FUNCTION_BLOCK FB_Cylinder IMPLEMENTS I_Cylinder
VAR_INPUT
	bAtBasePos		AT %I*	: BOOL;		// Hardware input signal: cylinder is at base position
	bAtWorkPos		AT %I*	: BOOL;		// Hardware input signal: cylinder is at work position
END_VAR
VAR_OUTPUT
	bMoveToWork		AT %Q*	: BOOL;		// Hardware output signal to move cylinder to work position
END_VAR

// =========================================================
;
// =========================================================

PROPERTY PUBLIC bState_AtBasePos : BOOL
GET
bState_AtBasePos := bAtBasePos;
END_GET
END_PROPERTY

PROPERTY PUBLIC bState_AtWorkPos : BOOL
GET
bState_AtWorkPos := bAtWorkPos;
END_GET
END_PROPERTY

PROPERTY PUBLIC bState_MoveToWork : BOOL
GET
bState_MoveToWork := bMoveToWork;
END_GET
END_PROPERTY

METHOD MoveToBase
VAR_INPUT
END_VAR
// =========================================================
	
StateMachine(	bBasePosReq := TRUE,
				bWorkPosReq	:= FALSE );
							
// =========================================================
END_METHOD

METHOD MoveToWork
VAR_INPUT
END_VAR
// =========================================================
	
StateMachine(	bBasePosReq := FALSE,
				bWorkPosReq	:= TRUE );
								
// =========================================================
END_METHOD

METHOD Reset
VAR_INPUT
END_VAR
// =========================================================

bMoveToWork := FALSE;

// =========================================================
END_METHOD

METHOD PROTECTED StateMachine
VAR_INPUT
	bBasePosReq		: BOOL;
	bWorkPosReq		: BOOL;
END_VAR
// =========================================================
// Base or work position requested
		
	IF bWorkPosReq THEN
		bMoveToWork := TRUE;
	END_IF
	
	IF bBasePosReq OR NOT bWorkPosReq THEN
		bMoveToWork := FALSE;
	END_IF

// =========================================================
END_METHOD

END_FUNCTION_BLOCK

// ---- 01_Submodules/Cylinder/POUs/FB_CylinderDiag.TcPOU
(* FB_CylinderDiag	- number of control signals:
							one direction is controllable
					- type of feedback signal:
							feedback in base and work position
					- with position diagnosis						*)
					
FUNCTION_BLOCK FB_CylinderDiag EXTENDS FB_Cylinder
VAR_INPUT
	tTimeOut 	 		: TIME;					// Time for watchdog that monitores if cylinder reaches base/work position
	fVibrationSensor	AT %I*	: LREAL;		// Hardware input signal: cylinder vibration
	fPressureSensor		AT %I*	: LREAL;		// Hardware input signal: cylinder pressure
END_VAR
VAR_OUTPUT
	bError				: BOOL;			// Error signal (diagnosed from position watchdog)
	sErrorMsg			: STRING;		// Error message
END_VAR
VAR
	fbTriggerError		: R_TRIG;		// Trigger to recognize rising edge of error
	bErrorMove			: BOOL;			// Move error
	fbTimerWatchDog		: TON;			// Watchdog timer for monitoring if cylinder reaches base/work position
END_VAR

// =========================================================
;
// =========================================================

METHOD PROTECTED Diag
VAR_INPUT
END_VAR
// =========================================================
// Timer starts when cylinder is not in base and work position
	
	IF NOT bAtBasePos AND NOT bAtWorkPos THEN
		fbTimerWatchDog(IN := TRUE,
						PT := tTimeOut);
	ELSE
		fbTimerWatchDog(IN := FALSE,
						PT := tTimeOut);
	END_IF

// =========================================================
// Error if cylinder does not reach base or work position
	
	fbTriggerError(CLK := fbTimerWatchDog.Q);
	
	bError := fbTimerWatchDog.Q;
	
	IF fbTriggerError.Q THEN
		bErrorMove := bMoveToWork;
	END_IF
	
	IF bError THEN
		IF bErrorMove = bMoveToWork THEN
			IF bMoveToWork THEN
				sErrorMsg := 'Work position not reached';
			ELSE
				sErrorMsg := 'Base position not reached';
			END_IF
		ELSE
			bError := FALSE;
			sErrorMsg := '';
		END_IF
	ELSE
		sErrorMsg := '';
	END_IF

// =========================================================
END_METHOD

METHOD Reset
VAR_INPUT
END_VAR
// =========================================================

// Calling method Reset of base class FB_Cylinder via 'SUPER^.'
SUPER^.Reset();		

// Reset error
bError 		:= FALSE;
sErrorMsg 	:= '';

// =========================================================
END_METHOD

METHOD PROTECTED StateMachine
VAR_INPUT
	bBasePosReq		: BOOL;
	bWorkPosReq		: BOOL;
END_VAR
// =========================================================

IF NOT bError THEN
	// Calling method StateMachine of base class FB_Cylinder via 'SUPER^.'
	SUPER^.StateMachine(bBasePosReq := bBasePosReq,
						bWorkPosReq	:= bWorkPosReq );
	
	// Diagnosis
	Diag();
END_IF

// =========================================================
END_METHOD

END_FUNCTION_BLOCK

// ---- 01_Submodules/Cylinder/POUs/FB_CylinderTemp.TcPOU
(* FB_CylinderTemp	- number of control signals:
							one direction is controllable
					- type of feedback signal:
							feedback in base and work position
					- with temperature signal					*)

FUNCTION_BLOCK FB_CylinderTemp EXTENDS FB_Cylinder
VAR_INPUT
	fTempCurrent	AT %I*	: LREAL;		// Hardware input signal: cylinder temperature
END_VAR

// =========================================================
;
// =========================================================

END_FUNCTION_BLOCK

// ---- 01_Submodules/Cylinder/POUs/FB_CylinderTempDiag.TcPOU
(* FB_CylinderTempDiag		- number of control signals:
									one direction is controllable
							- type of feedback signal:
									feedback in base and work position
							- with temperature diagnosis					*)

FUNCTION_BLOCK FB_CylinderTempDiag EXTENDS FB_CylinderTemp
VAR_INPUT
	fTempMax		AT %I*	: LREAL;		// Global input signal: maximal allowed cylinder temperature for temperature monitoring
	fTempMin		AT %I*	: LREAL;		// Global input signal: minimal allowed cylinder temperature for temperature monitoring
END_VAR
VAR_OUTPUT
	bError					: BOOL;			// Error signal (diagnosed from temperature monitoring)
	sErrorMsg				: STRING;		// Error message
END_VAR

// =========================================================
;
// =========================================================

METHOD PROTECTED StateMachine
VAR_INPUT
	bBasePosReq		: BOOL;
	bWorkPosReq		: BOOL;
END_VAR
// =========================================================

IF NOT bError THEN
	// Calling method StateMachine of base class FB_Cylinder via 'SUPER^.'
	SUPER^.StateMachine(bBasePosReq := bBasePosReq,
						bWorkPosReq	:= bWorkPosReq );
	
	// Diagnosis
	Diag();
END_IF

// =========================================================
END_METHOD

METHOD Reset
VAR_INPUT
END_VAR
// =========================================================
	
// Calling method Reset of base class FB_Cylinder via 'SUPER^.'
SUPER^.Reset();			

// Reset error
bError 		:= FALSE;
sErrorMsg 	:= '';

// =========================================================
END_METHOD

METHOD PROTECTED Diag
VAR_INPUT
END_VAR
// =========================================================
// Error if temperatur of cylinder is not in accepted interval
	
	bError := NOT (fTempCurrent >= fTempMin AND fTempCurrent <= fTempMax);
	
	IF bError THEN
		IF fTempCurrent > fTempMax THEN
			sErrorMsg := 'Temperature above maximum';
		ELSE
			sErrorMsg := 'Temperature below minimum';
		END_IF
	ELSE
		sErrorMsg := '';
	END_IF

// =========================================================
END_METHOD

END_FUNCTION_BLOCK

// ---- 01_Submodules/Cylinder/POUs/FB_CylinderTempRecord.TcPOU
(* FB_CylinderTempRecord	- number of control signals:
									one direction is controllable
							- type of feedback signal:
									feedback in base and work position
							- with temperature recording for data analysis		*)

FUNCTION_BLOCK FB_CylinderTempRecord EXTENDS FB_CylinderTemp
VAR_INPUT
	bRecordStart		: BOOL;						// Signal to start the temperature recording
	tIntervalTime		: TIME;						// Time of intervals to record the temperature 
END_VAR
VAR_OUTPUT
	bRecordDone			: BOOL;						// True if the temperature recording is done
	aTemps				: ARRAY[1..100] OF LREAL;	// Array with recorded temperatures
END_VAR
VAR
	fbTimerInterval		: TON;						// Timer to control the recording interval
	nIndex				: INT;						// Index to handle temperature array
END_VAR

// =========================================================
;
// =========================================================

METHOD Record
VAR_INPUT
END_VAR
// =========================================================
// Recording array filled
	
	bRecordDone := (nIndex = 100);

// =========================================================
// Recording temperatures
	
	IF bRecordStart AND NOT bRecordDone AND NOT fbTimerInterval.Q THEN
		fbTimerInterval(IN := TRUE,
						PT := tIntervalTime );
	END_IF
	
	IF fbTimerInterval.Q THEN
		fbTimerInterval(IN := FALSE);
		
		nIndex 			:= nIndex + 1;
		aTemps[nIndex] 	:= fTempCurrent;
	END_IF

// =========================================================
END_METHOD

METHOD Reset
VAR_INPUT
END_VAR
// =========================================================

// Calling method Reset of base class FB_Cylinder via 'SUPER^.'
SUPER^.Reset();

// Reset temperature array
FOR nIndex := 1 TO 100 BY 1 DO
	aTemps[nIndex] := 0;
END_FOR

// Reset index
nIndex := 0;

// =========================================================
END_METHOD

END_FUNCTION_BLOCK

// ---- 02_Subsystems/FB_SortingModule.TcPOU
// Module to select via sensor, cylinder and axis
FUNCTION_BLOCK FB_SortingModule EXTENDS FB_Subsystem_Root
VAR_INPUT
	// =============== Cylinder buttons =============================================
	bButtonCylToWorkIn			: BOOL;							// Signal of button to move cylinder to work position
	bButtonCylToBaseIn			: BOOL;							// Signal of button to move cylinder to base position
END_VAR
VAR_OUTPUT
	// =============== Process information ==========================================
	bSelected					: BOOL;							// Gets true if one sorting process is done
	
	// =============== For movement simulation on visualization =====================
	bCylinderToWork				: BOOL;							// Simulation of cylinder movement to work position
	
	// =============== Error variables ==============================================
	bCylError					: BOOL;							// Error signal of cylinder
	sCylErrorMsg				: STRING;						// Error message of cylinder
	
	// =============== Temperature recording ========================================
	aTemps						: ARRAY[1..100] OF LREAL;		// Array with recorded temperatures of cylinder
	
	// =============== Button return signals ========================================
	bButtonCylToWorkOut			: BOOL;							// Processed signal for button to move cylinder to work position
	bButtonCylToBaseOut			: BOOL;							// Processed signal for button to move cylinder to base position
END_VAR
VAR
	// =============== Function block instance of sensor ============================	
	fbSensorDelay				: FB_SignalHandlingDelay;		// Sensor needed for sorting process
	
	// =============== Function block instances for cylinder ========================
	fbCylinder					: FB_Cylinder;					// Without diagnosis and temperature mode
	fbCylinderDiag				: FB_CylinderDiag;				// With diagnosis of states
	fbCylinderTemp				: FB_CylinderTemp;				// With temperature mode
	fbCylinderTempDiag			: FB_CylinderTempDiag;			// With diagnosis of temperature
	fbCylinderTempRecord		: FB_CylinderTempRecord;		// With record of temperatures
	
	// =============== Interface instance for cylinder ==============================
	ipCylinder					: I_Cylinder;					// Interface for flexible access to cylinder FBs
	
	// =============== Submodule parameters =========================================
	tTimeOutCylinder			: TIME;							// For cylinder with diagnosis: time in which the cylinder should reach base/work position
	tRecordIntervalCylinder		: TIME;							// Time of intervals to record the temperature of cylinder
	tSensorDelay				: TIME;							// Time to delay sensor signal (time between hardware and processed software signal)
	tMoveAxis					: TIME;							// Time to move axis
	
	// =============== Manual cylinder control ======================================
	fbButtonCylToWork			: FB_SignalHandlingIntern;		// To move cylinder manually to work position
	fbButtonCylToBase			: FB_SignalHandlingIntern;		// To move cylinder manually to base position

	// =============== Common variables =============================================
	fbTimerAxis					: TON;							// Timer to move axis in (semi) automatic mode	
	fbTriggerCylAtWork			: R_TRIG;						// Trigger to recognize rising edge of cylinder being at work position
	eStateAutoAxis				: E_StateSortingAutoAxis;		// State variable for automatic mode - process to move axis
	eStateAutoCylinder			: E_StateSortingAutoCylinder;	// State variable for automatic mode - process to move cylinder
END_VAR

// =========================================================
;
// =========================================================

METHOD Automatic
VAR_INPUT
END_VAR
// =========================================================
// Process of sorting boxes - axis movement

	fbTriggerCylAtWork(CLK := ipCylinder.bState_AtWorkPos);			// Accessing property of FB via interface instance

	CASE eStateAutoAxis OF
		
		// =========================================================
		E_StateSortingAutoAxis.WaitForCylinderAtWorkPos:
		
						IF fbTriggerCylAtWork.Q THEN
							fbTimerAxis(IN := TRUE,
										PT := tMoveAxis);
										
							eStateAutoAxis := E_StateSortingAutoAxis.MoveAxis;
						END_IF
		
		// =========================================================
		E_StateSortingAutoAxis.MoveAxis:
		
						fbTimerAxis();
						
						IF bHaltRequest THEN
							eStateAutoAxis := E_StateSortingAutoAxis.StopAxis;
						ELSIF fbTimerAxis.Q THEN
							fbTimerAxis(IN := FALSE);
							
							bSelected 		:= TRUE;
							eStateAutoAxis	:= E_StateSortingAutoAxis.StopAxis;
						ELSE
							fbAxis.MoveFw();
						END_IF
		
		
		// =========================================================
		E_StateSortingAutoAxis.StopAxis:
		
						bSelected := FALSE;
						
						IF NOT bHaltDone THEN
							Stop(bHalt := TRUE);
						ELSE
							Stop(bHalt := FALSE);
							
							eStateAutoAxis := E_StateSortingAutoAxis.WaitForCylinderAtWorkPos;
						END_IF
	END_CASE
	
// =========================================================
// Process of sorting boxes - cylinder movement

	CASE eStateAutoCylinder OF
		
		// =========================================================
		// Detecting a box
		E_StateSortingAutoCylinder.DetectBox:	
		
					ipCylinder.MoveToBase();								// Calling method of FB via interface instance
					
					IF fbSensorDelay.bOut THEN
						eStateAutoCylinder := E_StateSortingAutoCylinder.CylToWork;
					END_IF
			
		// =========================================================
		// Moving cylinder to work position
		E_StateSortingAutoCylinder.CylToWork:
		
					ipCylinder.MoveToWork();								// Calling method of FB via interface instance
					
					IF ipCylinder.bState_AtWorkPos THEN					// Accessing property of FB via interface instance
						eStateAutoCylinder := E_StateSortingAutoCylinder.CylToBase;
					END_IF
		
		// =========================================================
		// Moving cylinder back to base position
		E_StateSortingAutoCylinder.CylToBase:
		
					ipCylinder.MoveToBase();								// Calling method of FB via interface instance
					
					IF ipCylinder.bState_AtBasePos THEN					// Accessing property of FB via interface instance
						eStateAutoCylinder := E_StateSortingAutoCylinder.DetectBox;
					END_IF
	END_CASE

// =========================================================
END_METHOD

PROPERTY bState_CylinderAtBasePos : BOOL
GET
bState_CylinderAtBasePos := ipCylinder.bState_AtBasePos;
END_GET
END_PROPERTY

PROPERTY bState_CylinderAtWorkPos : BOOL
GET
bState_CylinderAtWorkPos := ipCylinder.bState_AtWorkPos;
END_GET
END_PROPERTY

METHOD CylinderOptions
VAR_INPUT
	bCylinderDiag		: BOOL;		// If true the cylinder has diagnosis functionality
	bCylinderTemp		: BOOL;		// IF true the cylinder has temperature functionality
	bCylinderRecord		: BOOL;		// If true the cylinder has recording functionality
END_VAR
// =========================================================
// Selecting cylinder

	// Checking variables to enable/disable diagnosis and temperature mode
	IF bCylinderDiag THEN
		IF bCylinderTemp THEN
			// ============== FB with diagnosis and temperature mode ==============
			bCylError 		:= fbCylinderTempDiag.bError;						// Assigning output variable of chosen FB to local output variable
			sCylErrorMsg 	:= fbCylinderTempDiag.sErrorMsg;
			ipCylinder		:= fbCylinderTempDiag;								// Assigning chosen FB instance to interface instance
		
		ELSE
			// ============== FB with diagnosis and without temperature mode ==============
			fbCylinderDiag.tTimeOut 	:= tTimeOutCylinder;					// Setting special data for selected FB
			bCylError 					:= fbCylinderDiag.bError;				// Assigning output variable of chosen FB to local output variable
			sCylErrorMsg 				:= fbCylinderDiag.sErrorMsg;		
			ipCylinder					:= fbCylinderDiag;						// Assigning chosen FB instance to interface instance
		END_IF
		
	ELSE
		bCylError 		:= FALSE;
		sCylErrorMsg 	:= '';
		
		IF bCylinderTemp THEN
			IF bCylinderRecord THEN
				// ============== FB without diagnosis and with temperature recording ==============
				fbCylinderTempRecord.tIntervalTime	:= tRecordIntervalCylinder;	// Time of record interval
				fbCylinderTempRecord.bRecordStart 	:= bComprAirEnabledLocal;	// Recording if compressed air is set
				
				fbCylinderTempRecord.Record();									// Calling method of function block FB_CylinderTempRecord
				
				aTemps		:= fbCylinderTempRecord.aTemps;						// Saving output variable
				ipCylinder 	:= fbCylinderTempRecord;							// Assigning chosen FB instance to interface instance
			ELSE
				// ============== FB without diagnosis and with temperature mode, but without recording ==============
				ipCylinder 	:= fbCylinderTemp; 									// Assigning chosen FB instance to interface instance
			END_IF
			
		ELSE
			// ============== FB without diagnosis and without temperature mode ==============
			ipCylinder := fbCylinder;											// Assigning chosen FB instance to interface instance					
		END_IF	
	END_IF
									
// =========================================================
END_METHOD

METHOD Enable
VAR_INPUT
	bComprAirEnabled		: BOOL;			// Enable of compressed air
	bAxisEnable				: BOOL;			// Enable of axis
	bSensorEnable			: BOOL;			// Enable of sensor
	bManualAxisEnable		: BOOL;			// Enable of manual axis control
END_VAR
// =========================================================
// Calling method Enable of base class FB_Module via 'SUPER^.'
		
	SUPER^.Enable(	bComprAirEnabled	:= bComprAirEnabled,
					bAxisEnable			:= bAxisEnable,
					bSensorEnable		:= bSensorEnable,
					bManualAxisEnable	:= bManualAxisEnable);

// =========================================================
// Sensor control
		
	fbSensorDelay.Enable(bEnable := bSensorEnable);

// =========================================================
// Cylinder control (accessing property of FB via interfaces intance)
		
	fbButtonCylToWork.Enable(bEnable := bManualCylinderEnable AND NOT ipCylinder.bState_AtWorkPos);
	fbButtonCylToBase.Enable(bEnable := bManualCylinderEnable AND NOT ipCylinder.bState_AtBasePos);
	
	fbButtonCylToBase.bInput := NOT fbButtonCylToWork.bInput;

// =========================================================
END_METHOD

METHOD InputOutput
VAR_INPUT
END_VAR
// =========================================================
// Calling method SetOutput of base class FB_Module via 'SUPER^.'
		
	SUPER^.InputOutput();

// =========================================================
// Sensor
		
	fbSensorDelay.SetOutput();

// =========================================================
// Cylinder buttons
		
	fbButtonCylToWork.SetOutput();
	fbButtonCylToBase.SetOutput();

// =========================================================
// Output variables for cylinder
		
	bCylinderToWork := ipCylinder.bState_MoveToWork;		// Accessing property of selected FB via interface instance

// =========================================================
// Buttons
		
	fbButtonCylToWork.bInput 	:= bButtonCylToWorkIn;
	fbButtonCylToBase.bInput	:= bButtonCylToBaseIn;
	bButtonCylToWorkOut 		:= fbButtonCylToWork.bOut;
	bButtonCylToBaseOut 		:= fbButtonCylToBase.bOut;

// =========================================================
END_METHOD

METHOD Maintenance
VAR_INPUT
END_VAR
// =========================================================
// Calling own method Manual of this class FB_SortingModule via 'THIS^.'
		
	THIS^.Manual();

// =========================================================
END_METHOD

METHOD Manual
VAR_INPUT
END_VAR
// =========================================================
// Calling method Manual of base class FB_Module via 'SUPER^.'
		
	SUPER^.Manual();

// =========================================================
// Manual cylinder control (Calling methods of FB via interface instance)
	
	// Cylinder to work position
	IF fbButtonCylToWork.bOut THEN
		ipCylinder.MoveToWork();
	// Cylinder to base position
	ELSIF fbButtonCylToBase.bOut THEN
		ipCylinder.MoveToBase();
	END_IF

// =========================================================
END_METHOD

METHOD Reset
VAR_INPUT
	bReset		: BOOL;				// True if machine is in state RESETTING
END_VAR
// =========================================================
// Calling action Reset of base class FB_Module via 'SUPER^.'
		
	SUPER^.Reset(bReset := bReset);

// =========================================================
// Resetting cylinder and axis
	
	IF fbTriggerResetStart.Q THEN
		bSelected := FALSE;
		
		fbTimerAxis(IN := FALSE);
		
		// Calling method of FB via interface instance
		ipCylinder.Reset();
	END_IF

// =========================================================
END_METHOD

METHOD PROTECTED ResetState
VAR_INPUT
END_VAR
// =========================================================

eStateAutoAxis		:= E_StateSortingAutoAxis.WaitForCylinderAtWorkPos;
eStateAutoCylinder 	:= E_StateSortingAutoCylinder.DetectBox;

// =========================================================
END_METHOD

METHOD Semiautomatic
VAR_INPUT
END_VAR
// =========================================================
// Calling own method Automatic of this class FB_SortingModule via 'THIS^.'
		
	THIS^.Automatic();				

// =========================================================
END_METHOD

METHOD Starting
VAR_INPUT
	bStarting		: BOOL;			// True if machine is in state STARTING
END_VAR
// =========================================================
// Setting time to delay sensor
		
	fbSensorDelay.tDelay := tSensorDelay;

// =========================================================
// Calling method Starting of base class FB_Module via 'SUPER^.'
		
	SUPER^.Starting(bStarting := bStarting);

// =========================================================
END_METHOD

PROPERTY tAxisMovement : TIME
GET
tAxisMovement := tMoveAxis;
END_GET
SET
tMoveAxis := tAxisMovement;
END_SET
END_PROPERTY

PROPERTY tDelayOfSensor : TIME
GET
tDelayOfSensor := tSensorDelay;
END_GET
SET
tSensorDelay := tDelayOfSensor;
END_SET
END_PROPERTY

PROPERTY tRecordIntervalOfCylinder : TIME
GET
tRecordIntervalOfCylinder := tRecordIntervalCylinder;
END_GET
SET
tRecordIntervalCylinder := tRecordIntervalOfCylinder;
END_SET
END_PROPERTY

PROPERTY tTimeOutOfCylinder : TIME
GET
tTimeOutOfCylinder := tTimeOutCylinder;
END_GET
SET
tTimeOutCylinder := tTimeOutOfCylinder;
END_SET
END_PROPERTY

END_FUNCTION_BLOCK

// ---- 01_Submodules/Signal handling/POUs/FB_SignalHandlingDelay.TcPOU
FUNCTION_BLOCK FB_SignalHandlingDelay EXTENDS FB_SignalHandling
VAR_INPUT
	tDelay				: TIME;			// Time to delay input signal (time between hardware and processed software signal)
END_VAR
VAR
	bStartProcessing	: BOOL;			// To start the processing/delay of input signal
	fbTimerDelay		: TON;			// Timer to control the processing/delay of input signal
END_VAR

// =========================================================
;
// =========================================================

METHOD SetOutput
VAR_INPUT
END_VAR
// =========================================================

IF bEnableLocal AND bInput THEN
	bStartProcessing := TRUE;
END_IF

IF bStartProcessing THEN
	fbTimerDelay(	IN := TRUE,
					PT := tDelay);
ELSE
	fbTimerDelay(	IN := FALSE);
END_IF

IF fbTimerDelay.Q THEN
	bStartProcessing := FALSE;
	
	fbTimerDelay(IN := FALSE);
	
	bOut := TRUE;
ELSE
	bOut := FALSE;
END_IF
			
// =========================================================
END_METHOD

END_FUNCTION_BLOCK

// ---- 05_Visu/FB_Visu.TcPOU
FUNCTION_BLOCK FB_Visu
VAR_INPUT
	// =============== Sensors to detect boxes ==================
	bBarrierSensor			AT %I*	: BOOL;						// True if barrier sensor detects a box
	bMetalSensor			AT %I*	: BOOL;						// True if metal sensor detects a metal box
	bPlasticSensor			AT %I*	: BOOL;						// True if plastic sensor detects a box
	
	// =============== Axis =====================================
	fAxisVelo						: LREAL;					// Axis velocity
	
	// =============== State of machine elements ================
	bComprAirEnabled				: BOOL;						// True if compressed air is enabled
	bPowerEnabled					: BOOL;						// True if power supply is enabled
	bMainAxisMoves					: BOOL;						// True if main axis is moving
	bMetalAxisMoves					: BOOL;						// True if metal axis is moving
	bPlasticAxisMoves				: BOOL;						// True if plastic axis is moving
	bClampToWork					: BOOL;						// True if clamp cylinder moves to work position
	bBarrierToWork					: BOOL;						// True if barrier cylinder moves to work position
	bMetalToWork					: BOOL;						// True if metal cylinder moves to work position
	bPlasticToWork					: BOOL;						// True if plastic cylinder moves to work position
	
	// =============== Error ====================================
	bError							: BOOL;						// True if modules have errors
	bClampError						: BOOL;						// True if clamp cylinder has an error
	sClampErrMsg					: STRING;					// Error message of clamp cylinder
	bMetalCylError					: BOOL;						// True if metal cylinder has an error
	sMetalErrMsg					: STRING;					// Error message of metal cylinder
	bPlasticCylError				: BOOL;						// True if plastic cylinder has an error
	sPlasticErrMsg					: STRING;					// Error message of plastic cylinder
	nMainAxisErrorId				: UDINT;					// Error id of main axis
	nMetalAxisErrorId				: UDINT;					// Error id of metal axis
	nPlasticAxisErrorId				: UDINT;					// Error id of plastic axis
	
	// =============== PS_PackML_StateMachine ===================
	bStarted						: BOOL;						// True if state machine is in state EXECUTE
	bStopped						: BOOL;						// True if state machine is in state STOPPED
	bReset							: BOOL;						// True if state machine is in state RESETTING
	bAborted						: BOOL;						// True if state machine is in state ABORTED
	bIdle							: BOOL;						// True if state machine is in state IDLE
	bAuto							: BOOL;						// True if state machine is in mode AUTOMATIC
	bSemi							: BOOL;						// True if state machine is in mode SEMIAUTOMATIC
	bManual							: BOOL;						// True if state machine is in mode MANUAL
	bMaintenance					: BOOL;						// True if state machine is in mode MAINTENANCE
	bStartButtonOff					: BOOL;						// To turn off start button

	// =============== Buttons of visualization - inputs ========
	// State buttons
	bButtonPowerIn					: BOOL;						// Input signal of power button
	bButtonComprAirIn				: BOOL;						// Input signal of compressed air button
	bButtonStartIn					: BOOL;						// Input signal of start button
	bButtonStopIn					: BOOL;						// Input signal of stop button
	bButtonResetIn					: BOOL;						// Input signal of reset button
	bButtonAbortIn					: BOOL;						// Input signal of abort button
	
	// Mode buttons
	bButtonAutoIn					: BOOL;						// Input signal of automatic button
	bButtonSemiIn					: BOOL;						// Input signal of semi-automatic button
	bButtonManuIn					: BOOL;						// Input signal of manual button
	bButtonMaintenanceIn			: BOOL;						// Input signal of maintenance button
	
	// Axis buttons
	bButtonMainFwIn					: BOOL;						// Input signal of button to move main axis forwards
	bButtonMainBwIn					: BOOL;						// Input signal of button to move main axis backwards
	bButtonMetalFwIn				: BOOL;						// Input signal of button to move metal axis forwards
	bButtonMetalBwIn				: BOOL;						// Input signal of button to move metal axis backwards
	bButtonPlasticFwIn				: BOOL;						// Input signal of button to move plastic axis forwards
	bButtonPlasticBwIn				: BOOL;						// Input signal of button to move plastic axis backwards
	
	// Cylinder buttons
	bButtonClampToWorkIn			: BOOL;						// Input signal of button to move clamp cylinder
	bButtonBarrierToWorkIn			: BOOL;						// Input signal of button to move barrier cylinder
	bButtonMetalToWorkIn			: BOOL;						// Input signal of button to move metal cylinder
	bButtonPlasticToWorkIn			: BOOL;						// Input signal of button to move plastic cylinder
END_VAR
VAR_OUTPUT
	fYClamp					AT %Q*	: LREAL;					// Y-Coordinate of clamp cylinder
	fYBarrier				AT %Q*	: LREAL;					// Y-Coordinate of barrier cylinder
	fYMetal					AT %Q*	: LREAL;					// Y-Coordinate of metal cylinder
	fYPlastic				AT %Q*	: LREAL;					// Y-Coordinate of plastic cylinder
	aBoxX					AT %Q*	: ARRAY[1..4] OF LREAL;		// X-Coordinates of boxes
	aBoxY					AT %Q*	: ARRAY[1..4] OF LREAL;		// Y-Coordinates of boxes
	
	// =============== Buttons of visualization - outputs =======
	// State buttons
	bButtonPowerOut					: BOOL;						// To turn on and off the machine
	bButtonComprAirOut				: BOOL;						// To enable compressed air
	bButtonStartOut					: BOOL;						// To change state into state START
	bButtonStopOut					: BOOL;						// To change state into state STOP
	bButtonResetOut					: BOOL;						// To change state into state RESET
	
	// Mode buttons
	bButtonAutoOut					: BOOL;						// To change mode into mode AUTOMATIC		
	bButtonSemiOut					: BOOL;						// To change mode into mode SEMI-AUTOMATIC	
	bButtonManuOut					: BOOL;						// To change mode into mode MANAUL	
	bButtonMaintenanceOut			: BOOL;						// To change mode into mode MAINTENANCE	
	
	// Axis buttons
	bButtonMainFwOut				: BOOL;						// To move main axis forwards
	bButtonMainBwOut				: BOOL;						// To move main axis backwards
	bButtonMetalFwOut				: BOOL;						// To move metal axis forwards
	bButtonMetalBwOut				: BOOL;						// To move metal axis backwards
	bButtonPlasticFwOut				: BOOL;						// To move plastic axis forwards
	bButtonPlasticBwOut				: BOOL;						// To move plastic axis backwards
	
	// Cylinder buttons
	bButtonClampToWorkOut			: BOOL;						// To move manually clamp cylinder to work position
	bButtonBarrierToWorkOut			: BOOL;						// To move manually barrier cylinder to work position
	bButtonMetalToWorkOut			: BOOL;						// To move manually metal cylinder to work position
	bButtonPlasticToWorkOut			: BOOL;						// To move manually plastic cylinder to work position
END_VAR
VAR
	// =============== Boxes movement ===========================
	nLastBox						: INT;						// Box on last position of main belt
	aBoxMetalMove					: ARRAY[1..4] OF BOOL;		// bBoxMetalMove[1] is true, if box 1 is moved by metal cylinder
	aBoxMetalFree					: ARRAY[1..4] OF BOOL;		// bBoxMetalFree[1] is true, if any box blockades the movement of box 1 on metal belt
	aBoxPlasticMove					: ARRAY[1..4] OF BOOL;		// bBoxPlasticMove[1] is true, if box 1 is moved by plastic cylinder
	aBoxPlasticFree					: ARRAY[1..4] OF BOOL;		// bBoxMetalFree[1] is true, if any box blockades the plastic belt
	aBoxMainBelt					: ARRAY[1..4] OF BOOL;		// bBoxMainBelt[1] is true, if box 1 is on main belt and has no obstacles, so box 1 is moved by main axis
	aBoxMetalBelt					: ARRAY[1..4] OF BOOL;		// aBoxMetalBelt[1] is true, if box 1 is on metal belt and has no obstacles, so box 1 is moved by metal axis
	aBoxPlasticBelt					: ARRAY[1..4] OF BOOL;		// aBoxPlasticBelt[1] is true, if box 1 is on plastic belt and has no obstacles, so box 1 is moved by plastic axis
	fMainVelo						: LREAL;					// Velocity of boxes on main belt
	fMetalVelo						: LREAL;					// Velocity of boxes on metal belt
	fPlasticVelo					: LREAL;					// Velocity of boxes on plastic belt
	bAccident						: BOOL;						// True if machine caused an accident
	nState							: INT;
	
	// =============== Message ==================================
	nMessages						: INT;						// Number of messages
	sMessageClamp					: STRING;					// Message of clamp cylinder
	sMessageMetalCyl				: STRING;					// Message of metal cylinder
	sMessagePlasticCyl				: STRING;					// Message of plastic cylinder
	sMessageMainAxis				: STRING;					// Message of main axis
	sMessageMetalAxis				: STRING;					// Message of metal axis
	sMessagePlasticAxis				: STRING;					// Message of plastic axis
	
	// =============== Axes movement ============================
	nAngleMain						: INT;						// Angle of main axis element
	nAngleMetal						: INT;						// Angle of metal axis element
	nAnglePlastic					: INT;						// Angle of plastic axis element
	fbTimerMainAxis					: TON;						// Timer for movement of main axis element
	fbTimerMetalAxis				: TON;						// Timer for movement of metal axis element
	fbTimerPlasticAxis				: TON;						// Timer for movement of plastic axis element
	tMoveAxis						: TIME := T#40MS;			// Time for movement of elements

	// =============== Color variables ==========================
	nButtonColorStart				: DWORD;					// Color of start button
	bButtonColorStart				: BOOL;						// To change color of start button
	nButtonColorStop				: DWORD;					// Color of stop button
	bButtonColorStop				: BOOL;						// To change color of stop button
	nButtonColorReset				: DWORD;					// Color of reset button
	bButtonColorReset				: BOOL;						// To change color of reset button
	nButtonColorAuto				: DWORD;					// Color of automatic button
	bButtonColorAuto				: BOOL;						// To change color of automatic button
	nButtonColorSemi				: DWORD;					// Color of semi-automatic button
	bButtonColorSemi				: BOOL;						// To change color of semi-automatic button
	nButtonColorManu				: DWORD;					// Color of manual button
	bButtonColorManu				: BOOL;						// To change color of manual button
	nButtonColorMaint				: DWORD;					// Color of maintenance button
	bButtonColorMaint				: BOOL;						// To change color of maintenance button
	nButtonColorClamp				: DWORD;					// Color of button to move clamp cylinder
	bButtonColorClamp				: BOOL;						// To change color of clamp button
	nButtonColorBarrier				: DWORD;					// Color of button to move barrier cylinder
	bButtonColorBarrier				: BOOL;						// To change color of barrier button
	nButtonColorMetalCyl			: DWORD;					// Color of button to move metal cylinder
	bButtonColorMetalCyl			: BOOL;						// To change color of metal cylinder button
	nButtonColorPlasticCyl			: DWORD;					// Color of button to move plastic cylinder
	bButtonColorPlasticCyl			: BOOL;						// To change color of plastic cylinder button
	nButtonColorMainFw				: DWORD;					// Color of button to move main axis forwards
	bButtonColorMainFw				: BOOL;						// To change color of button to move main axis fw.
	nButtonColorMainBw				: DWORD;					// Color of button to move main axis backwards
	bButtonColorMainBw				: BOOL;						// To change color of button to move main axis bw.
	nButtonColorMetalFw				: DWORD;					// Color of button to move metal axis forwards
	bButtonColorMetalFw				: BOOL;						// To change color of button to move metal axis fw.
	nButtonColorMetalBw				: DWORD;					// Color of button to move metal axis backwards
	bButtonColorMetalBw				: BOOL;						// To change color of button to move metal axis bw.
	nButtonColorPlasticFw			: DWORD;					// Color of button to move plastic axis forwards
	bButtonColorPlasticFw			: BOOL;						// To change color of button to move plastic axis fw.
	nButtonColorPlasticBw			: DWORD;					// Color of button to move plastic axis backwards
	bButtonColorPlasticBw			: BOOL;						// To change color of button to move plastic axis bw.
	nButtonColorComprAir			: DWORD;					// Color of button to enable/disable compressed air
	bButtonColorComprAir			: BOOL;						// To change color of button to control compressed air
	
	// ================= PPM calc ===========================================
	ctTotalCtr						: CTU;
	ctMetalCtr						: CTU;
	arrTotal						: ARRAY[0..9] OF DINT;
	arrMetal						: ARRAY[0..9] OF DINT;
	tmrPpm							: TON;
	
END_VAR
VAR CONSTANT
	// =============== Colors ===============================================
	cYellow 									: DWORD	:= 16#00FFFF80;		// Color code for yellow
	cGreen 										: DWORD	:= 16#0080FF00;		// Color code for green
	cPink 										: DWORD	:= 16#00FF8080;		// Color code for pink
	
	// =============== Velocities ===========================================
	cVelocityDenominator						: LREAL := 250.0;			// Velocity of visualization is a fraction of real axis velocity
	cAxisMovementSemiPlusAuto					: INT 	:= 2;				// Axis movement per cycle in mode Automatic and Semi Autoamtic
	cAxisMovementManual							: INT 	:= 1;				// Axis movement per cycle in mode Manual
	cClampMovement								: LREAL := 0.1;				// Cylinder movement per cycle for clamp cylinder
	cBarrierMovement							: LREAL := 1.0;				// Cylinder movement per cycle for barrier cylinder
	cMetalPlasticCylMovement					: LREAL := 1.0;				// Cylinder movement per cycle for metal and plastic cylinder
	
	// =============== Barrier, clamp, metal, plastic cylinder ==============
	cYClampCylStartPos							: LREAL := 0.0;				// Y-start-position of clamp cylinder (where movement starts)
	cYClampCylEndPos							: LREAL := 3.0;				// Y-end-position of clamp cylinder (where movement ends)
	cYBarrierCylStartPos						: LREAL := 0.0;				// Y-start-position of barrier cylinder (where movement starts)
	cYBarrierCylEndPos							: LREAL := 63.0;			// Y-end-position of barrier cylinder (where movement ends)
	cYMetalPlasticCylStartPos					: LREAL := 0.0;				// Y-start-position of metal and plastic cylinder (where movement starts)
	cYMetalPlasticCylEndPos						: LREAL := -73.0;			// Y-end-position of metal and plastic cylinder (where movement ends)
	
	// =============== Widths, distances ====================================
	cBoxWidth									: LREAL := 60.0;			// Width of a box in the visu
	cBarrierWidth								: LREAL := 30.0;			// Width of the barrier cylinder in the visu
	cDiffBarrierToStartOfMetalCyl				: LREAL := 191.0;			// Difference on visu from barrier to start of metal cylinder
	cDiffBarrierToEndOfMetalCyl					: LREAL := 261.0;			// Difference on visu from barrier to end of metal cylinder
	cDiffBarrierToStartOfPlasticCyl				: LREAL := 441.0;			// Difference on visu from barrier to start of plastic cylinder
	cYMetalPlasticCylOnMainBelt					: LREAL := -9.0;			// Y-Position of metal and plastic cylinder reaching the main belt
	cYBoxesOnMetalPlasticBelt_min				: LREAL := -65.0;			// Minimal Y-Position of boxes when being on metal or plastic belt
	cYBoxesOnMetalPlasticBelt_max				: LREAL := -140.0;			// Maximal Y-Position of boxes when being on metal or plastic belt
	
	// =============== Positions of boxes - main belt =======================
	cYforAllBoxesOnMainBelt						: LREAL := -5.0;			// Y-Position of boxes being on main belt
	cYforAllBoxesNotOnMainBelt					: LREAL := -60.0;			// Y-Position of boxes not being on main belt
	
	cYforAllBoxesStartPosMainBelt				: LREAL := 0.0;				// Y-Position of boxes when being on first position of main belt
	cXforAllBoxesStartPosMainBelt				: LREAL := -240.0;			// X-Position of boxes when being on first position of main belt
	cXforAllBoxesLastPossiblePosMainBelt		: LREAL := 461.0;			// Last possible X-position of boxes on main belt
	
	cXforAllBoxesCorrectPushMetalCyl_min		: LREAL := 180;				// Minimal X-Position of boxes when being pushed by metal cylinder to metal belt 
	cXforAllBoxesCorrectPushMetalCyl_max		: LREAL := 211;				// Maximal X-Position of boxes when being pushed by metal cylinder to metal belt 
	cXforAllBoxesIncorrectPushMetalCyl_min		: LREAL := 131;				// Minimal X-Position of boxes when being pushed by metal cylinder, but not pushed to metal belt
	cXforAllBoxesIncorrectPushMetalCyl_max		: LREAL := 261;				// Maximal X-Position of boxes when being pushed by metal cylinder, but not pushed to metal belt
	
	cXforAllBoxesCorrectPushPlasticCyl_min		: LREAL := 430;				// Minimal X-Position of boxes when being pushed by plastic cylinder to plastic belt 
	cXforAllBoxesCorrectPushPlasticCyl_max		: LREAL := 461;				// Minimal X-Position of boxes when being pushed by plastic cylinder to plastic belt 
	cXforAllBoxesIncorrectPushPlasticCyl_min	: LREAL := 381;				// Minimal X-Position of boxes when being pushed by plastic cylinder, but not pushed to plastic belt
	
	// Box 1
	cXforBox1_MainBelt_Diff2to1_min				: LREAL := 0.001;			// Minimal distance from box 2 to box 1 so that box 1 can be moved on main belt
	cXforBox1_MainBelt_Diff2to1_max				: LREAL := 119.99999;		// Maximal distance from box 2 to box 1 so that box 1 can be moved on main belt
	cXforBox1_MainBelt_Diff3to1_min				: LREAL := 60.001;			// Minimal distance from box 3 to box 1 so that box 1 can be moved on main belt
	cXforBox1_MainBelt_Diff3to1_max				: LREAL := 179.99999;		// Maximal distance from box 3 to box 1 so that box 1 can be moved on main belt
	cXforBox1_MainBelt_Diff4to1_min				: LREAL := 120.001;			// Minimal distance from box 4 to box 1 so that box 1 can be moved on main belt
	cXforBox1_MainBelt_Diff4to1_max				: LREAL := 239.99999;		// Maximal distance from box 4 to box 1 so that box 1 can be moved on main belt
	
	// Box 2
	cXforBox2_MainBelt_Diff1to2_min				: LREAL := -0.00001;		// Minimal distance from box 1 to box 2 so that box 2 can be moved on main belt
	cXforBox2_MainBelt_Diff1to2_max				: LREAL := -119.999;		// Maximal distance from box 1 to box 2 so that box 2 can be moved on main belt
	cXforBox2_MainBelt_Diff3to2_min				: LREAL := 119.99999;		// Minimal distance from box 3 to box 2 so that box 2 can be moved on main belt
	cXforBox2_MainBelt_Diff3to2_max				: LREAL := 0.001;			// Maximal distance from box 3 to box 2 so that box 2 can be moved on main belt
	cXforBox2_MainBelt_Diff4to2_min				: LREAL := 179.99999;		// Minimal distance from box 4 to box 2 so that box 2 can be moved on main belt
	cXforBox2_MainBelt_Diff4to2_max				: LREAL := 60.001;			// Maximal distance from box 4 to box 2 so that box 2 can be moved on main belt

	// Box 3
	cXforBox3_MainBelt_Diff1to3_min				: LREAL := -60.00001;		// Minimal distance from box 1 to box 3 so that box 3 can be moved on main belt
	cXforBox3_MainBelt_Diff1to3_max				: LREAL := -179.999;		// Maximal distance from box 1 to box 3 so that box 3 can be moved on main belt
	cXforBox3_MainBelt_Diff2to3_min				: LREAL := -0.00001;		// Minimal distance from box 2 to box 3 so that box 3 can be moved on main belt
	cXforBox3_MainBelt_Diff2to3_max				: LREAL := -119.999;		// Maximal distance from box 2 to box 3 so that box 3 can be moved on main belt
	cXforBox3_MainBelt_Diff4to3_min				: LREAL := 119.99999;		// Minimal distance from box 4 to box 3 so that box 3 can be moved on main belt
	cXforBox3_MainBelt_Diff4to3_max				: LREAL := 0.001;			// Maximal distance from box 4 to box 3 so that box 3 can be moved on main belt
	
	// Box 4
	cXforBox4_MainBelt_Diff1to4_min				: LREAL := -120.00001;		// Minimal distance from box 1 to box 4 so that box 4 can be moved on main belt
	cXforBox4_MainBelt_Diff1to4_max				: LREAL := -239.999;		// Maximal distance from box 1 to box 4 so that box 4 can be moved on main belt
	cXforBox4_MainBelt_Diff2to4_min				: LREAL := -60.00001;		// Minimal distance from box 2 to box 4 so that box 4 can be moved on main belt
	cXforBox4_MainBelt_Diff2to4_max				: LREAL := -179.999;		// Maximal distance from box 2 to box 4 so that box 4 can be moved on main belt
	cXforBox4_MainBelt_Diff3to4_min				: LREAL := -0.00001;		// Minimal distance from box 3 to box 4 so that box 4 can be moved on main belt
	cXforBox4_MainBelt_Diff3to4_max				: LREAL := -119.999;		// Maximal distance from box 3 to box 4 so that box 4 can be moved on main belt
	
	// =============== Positions of boxes - metal belt ======================
	// Box 1
	cXforBox1OnMetalBelt_min					: LREAL := 240;				// Minimal X-Position of box 1 when being on metal belt
	cXforBox1OnMetalBelt_max					: LREAL := 271;				// Maximal X-Position of box 1 when being on metal belt
	// Box 2
	cXforBox2OnMetalBelt_min					: LREAL := 300;				// Minimal X-Position of box 2 when being on metal belt
	cXforBox2OnMetalBelt_max					: LREAL := 331;				// Maximal X-Position of box 2 when being on metal belt
	// Box 3
	cXforBox3OnMetalBelt_min					: LREAL := 360;				// Minimal X-Position of box 3 when being on metal belt
	cXforBox3OnMetalBelt_max					: LREAL := 391;				// Maximal X-Position of box 3 when being on metal belt
	// Box 4
	cXforBox4OnMetalBelt_min					: LREAL := 420;				// Minimal X-Position of box 4 when being on metal belt
	cXforBox4OnMetalBelt_max					: LREAL := 451;				// Maximal X-Position of box 4 when being on metal belt
	
	// =============== Positions of boxes - plastic belt ====================
	// Box 1
	cXforBox1OnPlasticBelt_min					: LREAL := 470;				// Minimal X-Position of box 1 when being on plastic belt
	cXforBox1OnPlasticBelt_max					: LREAL := 521;				// Maximal X-Position of box 1 when being on plastic belt
	// Box 2
	cXforBox2OnPlasticBelt_min					: LREAL := 530;				// Minimal X-Position of box 2 when being on plastic belt
	cXforBox2OnPlasticBelt_max					: LREAL := 581;				// Maximal X-Position of box 2 when being on plastic belt
	// Box 3
	cXforBox3OnPlasticBelt_min					: LREAL := 590;				// Minimal X-Position of box 3 when being on plastic belt
	cXforBox3OnPlasticBelt_max					: LREAL := 641;				// Maximal X-Position of box 3 when being on plastic belt
	// Box 4
	cXforBox4OnPlasticBelt_min					: LREAL := 650;				// Minimal X-Position of box 4 when being on plastic belt
	cXforBox4OnPlasticBelt_max					: LREAL := 701;				// Maximal X-Position of box 4 when being on plastic belt
END_VAR

// =========================================================
// Resetting visu
	
	IF bReset THEN
		Reset();
	END_IF

// =========================================================
// Because of the visualisation size, the boxes velocity is a fraction of the axis velocity
	
	IF bAuto OR bSemi OR bButtonMainFwIn THEN
		fMainVelo := (fAxisVelo / cVelocityDenominator);
	ELSIF bButtonMainBwIn THEN
		fMainVelo := -(fAxisVelo / cVelocityDenominator);
	END_IF
	
	IF bAuto OR bSemi OR bButtonMetalFwIn THEN
		fMetalVelo := -(fAxisVelo / cVelocityDenominator);
	ELSIF bButtonMetalBwIn THEN
		fMetalVelo := (fAxisVelo / cVelocityDenominator);
	END_IF
	
	IF bAuto OR bSemi OR bButtonPlasticFwIn THEN
		fPlasticVelo := -(fAxisVelo / cVelocityDenominator);
	ELSIF bButtonPlasticBwIn THEN
		fPlasticVelo := (fAxisVelo / cVelocityDenominator);
	END_IF

// =========================================================
// In case of accident the power button is turned off
	
	IF bAccident THEN
		IF bButtonPowerOut THEN
			bButtonPowerOut := FALSE;
		END_IF
		
		IF bStopped THEN
			bAccident := FALSE;
		END_IF
	END_IF

// =========================================================
// Visuazation functions

	// Rotation of axis elements
	AxisRotation();
	
	// Buttons, order of boxes, error messages
	ButtonSignals();
	ButtonColors();
	LastBox();
	ErrorMessages();
	
	// Motion of cylinders
	Barrier_Clamp_Cyl();
	Metal_Plastic_Cyl();
	
	// Motion of boxes
	AxisMoveBoxes();
	CylinderMoveBoxes();

// =========================================================

// ==========================================================
// part per min calculation
tmrPpm(IN:=(NOT tmrPpm.Q), PT:=T#60S);
IF tmrPpm.Q THEN
	MEMCPY(ADR(arrTotal[1]), ADR(arrTotal[0]), SIZEOF(DINT) * 9);
	MEMCPY(ADR(arrMetal[1]), ADR(arrMetal[0]), SIZEOF(DINT) * 9);
END_IF
ctTotalCtr(CU:=bMetalToWork OR bPlasticToWork, CV=>arrTotal[0], RESET:=tmrPpm.Q);
ctMetalCtr(CU:=bMetalToWork, CV=>arrMetal[0], RESET:=tmrPpm.Q);

// ===========================================================

METHOD PRIVATE AxisMoveBoxes
VAR_INPUT
END_VAR
// =========================================================
// Checking traction standby on main belt
// bBoxMainBelt[1] is true, if box 1 is on main belt and has no obstacles, so box 1 is moved by main axis
		
	aBoxMainBelt[1] := 	// box 1 on main belt
						aBoxY[1] >= cYforAllBoxesOnMainBelt	
						// not previous to box 2											
						AND (	(aBoxX[2] - aBoxX[1] - fMainVelo) >= cXforBox1_MainBelt_Diff2to1_max
							OR 	(aBoxX[2] - aBoxX[1] - fMainVelo) <= cXforBox1_MainBelt_Diff2to1_min
							OR 	aBoxY[2] < cYforAllBoxesNotOnMainBelt)
						// not previous to box 3	
						AND (	(aBoxX[3] - aBoxX[1] - fMainVelo) >= cXforBox1_MainBelt_Diff3to1_max
							OR 	(aBoxX[3] - aBoxX[1]- fMainVelo) <= cXforBox1_MainBelt_Diff3to1_min
							OR 	aBoxY[3] < cYforAllBoxesNotOnMainBelt)
						// not previous to box 4
						AND (	(aBoxX[4] - aBoxX[1] - fMainVelo) >= cXforBox1_MainBelt_Diff4to1_max
							OR 	(aBoxX[4] - aBoxX[1]- fMainVelo) <= cXforBox1_MainBelt_Diff4to1_min
							OR	aBoxY[4] < cYforAllBoxesNotOnMainBelt);
						
	aBoxMainBelt[2] := 	// box 2 on main belt
						aBoxY[2] >= cYforAllBoxesOnMainBelt
						// not previous to box 1											
						AND (	(aBoxX[1] - aBoxX[2] - fMainVelo) >= cXforBox2_MainBelt_Diff1to2_min 
							OR 	(aBoxX[1] - aBoxX[2] - fMainVelo) <= cXforBox2_MainBelt_Diff1to2_max 
							OR 	aBoxY[1] < cYforAllBoxesNotOnMainBelt)
						// not previous to box 3											
						AND (	(aBoxX[3] - aBoxX[2] - fMainVelo) >= cXforBox2_MainBelt_Diff3to2_min 
							OR 	(aBoxX[3] - aBoxX[2] - fMainVelo) <= cXforBox2_MainBelt_Diff3to2_max 
							OR 	aBoxY[3] < cYforAllBoxesNotOnMainBelt)
						// not previous to box 4											
						AND (	(aBoxX[4] - aBoxX[2] - fMainVelo) >= cXforBox2_MainBelt_Diff4to2_min 
							OR 	(aBoxX[4] - aBoxX[2] - fMainVelo) <= cXforBox2_MainBelt_Diff4to2_max 
							OR 	aBoxY[4] < cYforAllBoxesNotOnMainBelt);
	
	aBoxMainBelt[3] := 	// box 3 on main belt
						aBoxY[3] >= cYforAllBoxesOnMainBelt
						// not previous to box 1											
						AND (	(aBoxX[1] - aBoxX[3] - fMainVelo) >= cXforBox3_MainBelt_Diff1to3_min
							OR 	(aBoxX[1] - aBoxX[3] - fMainVelo) <= cXforBox3_MainBelt_Diff1to3_max
							OR 	aBoxY[1] < cYforAllBoxesNotOnMainBelt)
						// not previous to box 2											
						AND (	(aBoxX[2] - aBoxX[3] - fMainVelo) >= cXforBox3_MainBelt_Diff2to3_min
							OR 	(aBoxX[2] - aBoxX[3] - fMainVelo) <= cXforBox3_MainBelt_Diff2to3_max 
							OR 	aBoxY[2] < cYforAllBoxesNotOnMainBelt)
						// not previous to box 4											
						AND (	(aBoxX[4] - aBoxX[3] - fMainVelo) >= cXforBox3_MainBelt_Diff4to3_min
							OR 	(aBoxX[4] - aBoxX[3] - fMainVelo) <= cXforBox3_MainBelt_Diff4to3_max
							OR 	aBoxY[4] < cYforAllBoxesNotOnMainBelt);
						
	aBoxMainBelt[4] := 	// box 4 on main belt
						aBoxY[4] >= cYforAllBoxesOnMainBelt
						// not previous to box 1											
						AND (	(aBoxX[1] - aBoxX[4] - fMainVelo) >= cXforBox4_MainBelt_Diff1to4_min
							OR 	(aBoxX[1] - aBoxX[4] - fMainVelo) <= cXforBox4_MainBelt_Diff1to4_max
							OR 	aBoxY[1] < cYforAllBoxesNotOnMainBelt)
						// not previous to box 2											
						AND (	(aBoxX[2] - aBoxX[4] - fMainVelo) >= cXforBox4_MainBelt_Diff2to4_min
							OR 	(aBoxX[2] - aBoxX[4] - fMainVelo) <= cXforBox4_MainBelt_Diff2to4_max
							OR 	aBoxY[2] < cYforAllBoxesNotOnMainBelt)
						// not previous to box 3											
						AND (	(aBoxX[3] - aBoxX[4] - fMainVelo) >= cXforBox4_MainBelt_Diff3to4_min
							OR 	(aBoxX[3] - aBoxX[4] - fMainVelo) <= cXforBox4_MainBelt_Diff3to4_max
							OR 	aBoxY[3] < cYforAllBoxesNotOnMainBelt);
					
// =========================================================
// Motion of boxes on main belt - forwards
					
	IF bMainAxisMoves AND (bAuto OR bSemi OR bButtonMainFwIn) THEN
		FOR nState := 1 TO 4 BY 1 DO
			IF aBoxMainBelt[nState] THEN	
				// not previous to moving metal cylinder
				IF aBoxX[nState] >= (cBoxWidth*nState + cBarrierWidth) AND aBoxX[nState] < (cBoxWidth*nState + cDiffBarrierToEndOfMetalCyl - 1) THEN
					// Metal cylinder over main belt
					IF fYMetal <= cYMetalPlasticCylOnMainBelt THEN
						IF aBoxX[nState] < (cBoxWidth*nState + cDiffBarrierToStartOfMetalCyl - cBoxWidth + 0.25)
						AND aBoxX[nState] > (cBoxWidth*nState + cDiffBarrierToStartOfMetalCyl - cBoxWidth - 0.15) THEN
							aBoxX[nState] := cBoxWidth*nState + cDiffBarrierToStartOfMetalCyl - cBoxWidth;
						ELSIF aBoxX[nState] <= (cBoxWidth*nState + cDiffBarrierToStartOfMetalCyl - cBoxWidth - 0.15) THEN
							aBoxX[nState] := aBoxX[nState] + fMainVelo;
						END_IF
					// Metal cylinder not over main belt
					ELSE
						aBoxX[nState] := aBoxX[nState] + fMainVelo;
					END_IF
				END_IF
				
				// not previous to moving plastic cylinder
				IF aBoxX[nState] >= (cBoxWidth*nState + cDiffBarrierToEndOfMetalCyl - 1) THEN
					// Plastic cylinder over main belt
					IF fYPlastic <= cYMetalPlasticCylOnMainBelt THEN
						IF aBoxX[nState] < (cBoxWidth*nState + cDiffBarrierToStartOfPlasticCyl - cBoxWidth + 0.25)
						AND aBoxX[nState] > (cBoxWidth*nState + cDiffBarrierToStartOfPlasticCyl - cBoxWidth - 0.15) THEN
							aBoxX[nState] := cBoxWidth*nState + cDiffBarrierToStartOfPlasticCyl - cBoxWidth;
						ELSIF aBoxX[nState] <= (cBoxWidth*nState + cDiffBarrierToStartOfPlasticCyl - cBoxWidth - 0.15) THEN
							aBoxX[nState] := aBoxX[nState] + fMainVelo;
						END_IF
					// Plastic cylinder not over main belt
					ELSE
						aBoxX[nState] := aBoxX[nState] + fMainVelo;
					END_IF
				END_IF
				
				// barrier open and box 1 in the first place
				IF fYBarrier >= (cBoxWidth + 1) AND aBoxX[nState] >= cBoxWidth*(nState - 1) AND aBoxX[nState] <  (cBoxWidth*nState + cBarrierWidth) THEN
					IF aBoxX[nState] + fMainVelo < (cBoxWidth*nState + cBarrierWidth) THEN
						 aBoxX[nState] := aBoxX[nState] + fMainVelo;
					ELSIF aBoxX[nState] < (cBoxWidth*nState + cBarrierWidth) THEN
						aBoxX[nState] := (cBoxWidth*nState + cBarrierWidth);
					END_IF
				END_IF
				
				// not previous to clamp
				IF aBoxX[nState] + fMainVelo < -cBoxWidth*(3 - nState) THEN
					aBoxX[nState] := aBoxX[nState] + fMainVelo;
				ELSIF aBoxX[nState] < -cBoxWidth*(nState + 1) THEN
					aBoxX[nState] := -cBoxWidth*(nState + 1);
				END_IF
				
				// clamp open, not after clamp											
				IF fYClamp >= 1 AND aBoxX[nState] >= -cBoxWidth*(nState + 1) THEN
					IF aBoxX[nState] + fMainVelo < cBoxWidth*(nState - 1) THEN
						aBoxX[nState] := aBoxX[nState] + fMainVelo;
					ELSIF aBoxX[nState] < cBoxWidth*(nState - 1) THEN
						aBoxX[nState] := cBoxWidth*(nState - 1);
					END_IF
				END_IF
			END_IF
		END_FOR
	END_IF

// =========================================================
// Motion of boxes on main belt - backwards
	
	IF bMainAxisMoves AND bButtonMainBwIn THEN 
		FOR nState := 1 TO 4 BY 1 DO
			IF aBoxMainBelt[nState] THEN
				// not previous to moving metal cylinder
				IF aBoxX[nState] >= (cBoxWidth*nState + cBoxWidth + cBarrierWidth) AND aBoxX[nState] < (cBoxWidth*nState + cDiffBarrierToEndOfMetalCyl + 1) THEN
					IF NOT (aBoxX[nState] < (cBoxWidth*nState + cDiffBarrierToEndOfMetalCyl + 0.25)
					AND aBoxX[nState] > (cBoxWidth*nState + cDiffBarrierToEndOfMetalCyl - 0.15)
					AND fYMetal <= cYMetalPlasticCylOnMainBelt) THEN
						aBoxX[nState] := aBoxX[nState] + fMainVelo;
					ELSE
						aBoxX[nState] := cBoxWidth*nState + cDiffBarrierToEndOfMetalCyl;
					END_IF
				END_IF
				
				// not previous to moving plastic cylinder
				IF aBoxX[nState] >= (cBoxWidth*nState + cDiffBarrierToEndOfMetalCyl + 1) THEN
					aBoxX[nState] := aBoxX[nState] + fMainVelo;
				END_IF
				
				// not previous to moving barrier cylinder
				IF aBoxX[nState] > cBoxWidth*(nState - 1) AND aBoxX[nState] < (cBoxWidth*nState + cBoxWidth + cBarrierWidth) THEN
					IF NOT (aBoxX[nState] < (cBoxWidth*nState + cBarrierWidth + 0.25)
					AND aBoxX[nState] > (cBoxWidth*nState + cBarrierWidth - 0.15)
					AND fYBarrier < (cBoxWidth + 1)) THEN
						aBoxX[nState] := aBoxX[nState] + fMainVelo;
					ELSE
						aBoxX[nState] := cBoxWidth*nState + cBarrierWidth;
					END_IF
				END_IF
				
				// barrier open and box 1 after the first place
				IF fYBarrier >= (cBoxWidth + 1) AND aBoxX[nState] < cBoxWidth*(nState + 1) AND aBoxX[nState] > cBoxWidth*(nState - 1) THEN
					aBoxX[nState] := aBoxX[nState] + fMainVelo;
				END_IF	
				
				// clamp open, not previous to clamp											
				IF fYClamp >= 1 AND aBoxX[nState] <= cBoxWidth*(nState-1) AND aBoxX[nState] > -cBoxWidth*(3-nState) THEN
					aBoxX[nState] := aBoxX[nState] + fMainVelo;
				END_IF
				
				// not at the beginning of main belt
				IF aBoxX[nState] > -cBoxWidth*(4-nState) AND aBoxX[nState] <= -cBoxWidth*(3-nState) THEN
					aBoxX[nState] := aBoxX[nState] + fMainVelo;
				END_IF
			END_IF
		END_FOR	
	END_IF

// =========================================================
// =========================================================
// Checking traction standby on metal belt
	
	aBoxMetalBelt[1] := // box 1 on metal belt
						aBoxX[1] > cXforBox1OnMetalBelt_min AND aBoxX[1] <= cXforBox1OnMetalBelt_max
						// not previous to box 2											
						AND ((aBoxY[2] - aBoxY[1] - fMetalVelo) >= cBoxWidth OR (aBoxY[2] - aBoxY[1] - fMetalVelo) <= -cBoxWidth
							OR NOT (aBoxX[2] > cXforBox2OnMetalBelt_min AND aBoxX[2] <= cXforBox2OnMetalBelt_max))
						// not previous to box 3	
						AND ((aBoxY[3] - aBoxY[1]- fMetalVelo) >= cBoxWidth OR (aBoxY[3] - aBoxY[1]- fMetalVelo) <= -cBoxWidth
							OR NOT (aBoxX[3] > cXforBox3OnMetalBelt_min AND aBoxX[3] <= cXforBox3OnMetalBelt_max))
						// not previous to box 4
						AND ((aBoxY[4] - aBoxY[1]- fMetalVelo) >= cBoxWidth OR (aBoxY[4] - aBoxY[1]- fMetalVelo) <= -cBoxWidth
							OR NOT (aBoxX[4] > cXforBox4OnMetalBelt_min AND aBoxX[4] <= cXforBox4OnMetalBelt_max));	
						
	aBoxMetalBelt[2] := aBoxX[2] > cXforBox2OnMetalBelt_min AND aBoxX[2] <= cXforBox2OnMetalBelt_max										
						AND ((aBoxY[1] - aBoxY[2] - fMetalVelo) >= cBoxWidth OR (aBoxY[1] - aBoxY[2] - fMetalVelo) <= -cBoxWidth
							OR NOT (aBoxX[1] > cXforBox1OnMetalBelt_min AND aBoxX[1] <= cXforBox1OnMetalBelt_max))
						AND ((aBoxY[3] - aBoxY[2]- fMetalVelo) >= cBoxWidth OR (aBoxY[3] - aBoxY[2]- fMetalVelo) <= -cBoxWidth
							OR NOT (aBoxX[3] > cXforBox3OnMetalBelt_min AND aBoxX[3] <= cXforBox3OnMetalBelt_max))
						AND ((aBoxY[4] - aBoxY[2]- fMetalVelo) >= cBoxWidth OR (aBoxY[4] - aBoxY[2]- fMetalVelo) <= -cBoxWidth
							OR NOT (aBoxX[4] > cXforBox4OnMetalBelt_min AND aBoxX[4] <= cXforBox4OnMetalBelt_max));	
						
	aBoxMetalBelt[3] := aBoxX[3] > cXforBox3OnMetalBelt_min AND aBoxX[3] <= cXforBox3OnMetalBelt_max										
						AND ((aBoxY[1] - aBoxY[3] - fMetalVelo) >= cBoxWidth OR (aBoxY[1] - aBoxY[3] - fMetalVelo) <= -cBoxWidth
							OR NOT (aBoxX[1] > cXforBox1OnMetalBelt_min AND aBoxX[1] <= cXforBox1OnMetalBelt_max))
						AND ((aBoxY[2] - aBoxY[3]- fMetalVelo) >= cBoxWidth OR (aBoxY[2] - aBoxY[3]- fMetalVelo) <= -cBoxWidth
							OR NOT (aBoxX[2] > cXforBox2OnMetalBelt_min AND aBoxX[2] <= cXforBox2OnMetalBelt_max))
						AND ((aBoxY[4] - aBoxY[3]- fMetalVelo) >= cBoxWidth OR (aBoxY[4] - aBoxY[3]- fMetalVelo) <= -cBoxWidth
							OR NOT (aBoxX[4] > cXforBox4OnMetalBelt_min AND aBoxX[4] <= cXforBox4OnMetalBelt_max));	
						
	aBoxMetalBelt[4] := aBoxX[4] > cXforBox4OnMetalBelt_min AND aBoxX[4] <= cXforBox4OnMetalBelt_max										
						AND ((aBoxY[1] - aBoxY[4] - fMetalVelo) >= cBoxWidth OR (aBoxY[1] - aBoxY[4] - fMetalVelo) <= -cBoxWidth
							OR NOT (aBoxX[1] > cXforBox1OnMetalBelt_min AND aBoxX[1] <= cXforBox1OnMetalBelt_max))
						AND ((aBoxY[2] - aBoxY[4] - fMetalVelo) >= cBoxWidth OR (aBoxY[2] - aBoxY[4] - fMetalVelo) <= -cBoxWidth
							OR NOT (aBoxX[2] > cXforBox2OnMetalBelt_min AND aBoxX[2] <= cXforBox2OnMetalBelt_max))
						AND ((aBoxY[3] - aBoxY[4]- fMetalVelo) >= cBoxWidth OR (aBoxY[3] - aBoxY[4]- fMetalVelo) <= -cBoxWidth
							OR NOT (aBoxX[3] > cXforBox3OnMetalBelt_min AND aBoxX[3] <= cXforBox3OnMetalBelt_max));

// =========================================================
// Motion of boxes on metal belt and back to the start position number 4
	
	FOR nState := 1 TO 4 BY 1 DO	
		IF bMetalAxisMoves THEN
			IF 	aBoxMetalBelt[nState] THEN
					// Check the state and direction of motion		
					IF bAuto OR bSemi OR (NOT bAuto AND bButtonMetalFwIn) THEN
						// Move box to the end of metal belt and then back to position 4	
						IF aBoxY[nState] <= (cYBoxesOnMetalPlasticBelt_min + 0.1) AND aBoxY[nState] > cYBoxesOnMetalPlasticBelt_max THEN
							aBoxY[nState] := aBoxY[nState] + fMetalVelo;
						END_IF
						
					ELSIF NOT bAuto AND bButtonMetalBwIn THEN
						IF aBoxY[nState] + fMetalVelo <= (cYBoxesOnMetalPlasticBelt_min - 0.1) THEN
							aBoxY[nState] := aBoxY[nState] + fMetalVelo;
						END_IF
					END_IF
			END_IF
		END_IF	
		
		IF aBoxY[nState] <= cYBoxesOnMetalPlasticBelt_max AND nLastBox = 0 THEN
			aBoxY[nState] := cYforAllBoxesStartPosMainBelt;
			aBoxX[nState] := cXforAllBoxesStartPosMainBelt + nState*cBoxWidth;
		END_IF
	END_FOR
	
// =========================================================
// =========================================================
// Checking traction standby on plastic belt
	
	aBoxPlasticBelt[1] := // box 1 on plastic belt
						aBoxX[1] > cXforBox1OnPlasticBelt_min AND aBoxX[1] <= cXforBox1OnPlasticBelt_max	
						// not previous to box 2											
						AND ((aBoxY[2] - aBoxY[1] - fPlasticVelo) >= cBoxWidth OR (aBoxY[2] - aBoxY[1] - fPlasticVelo) <= -cBoxWidth
								OR NOT (aBoxX[2] > cXforBox2OnPlasticBelt_min AND aBoxX[2] <= cXforBox2OnPlasticBelt_max))
						// not previous to box 3	
						AND ((aBoxY[3] - aBoxY[1]- fPlasticVelo) >= cBoxWidth OR (aBoxY[3] - aBoxY[1]- fPlasticVelo) <= -cBoxWidth
								OR NOT (aBoxX[3] > cXforBox3OnPlasticBelt_min AND aBoxX[3] <= cXforBox3OnPlasticBelt_max))
						// not previous to box 4
						AND ((aBoxY[4] - aBoxY[1]- fPlasticVelo) >= cBoxWidth OR (aBoxY[4] - aBoxY[1]- fPlasticVelo) <= -cBoxWidth
								OR NOT (aBoxX[4] > cXforBox4OnPlasticBelt_min AND aBoxX[4] <= cXforBox4OnPlasticBelt_max));	
						
	aBoxPlasticBelt[2] := aBoxX[2] > cXforBox2OnPlasticBelt_min AND aBoxX[2] <= cXforBox2OnPlasticBelt_max									
						AND ((aBoxY[1] - aBoxY[2] - fPlasticVelo) >= cBoxWidth OR (aBoxY[1] - aBoxY[2] - fPlasticVelo) <= -cBoxWidth
								OR NOT (aBoxX[1] > cXforBox1OnPlasticBelt_min AND aBoxX[1] <= cXforBox1OnPlasticBelt_max))
						AND ((aBoxY[3] - aBoxY[2]- fPlasticVelo) >= cBoxWidth OR (aBoxY[3] - aBoxY[2]- fPlasticVelo) <= -cBoxWidth
								OR NOT (aBoxX[3] > cXforBox3OnPlasticBelt_min AND aBoxX[3] <= cXforBox3OnPlasticBelt_max))
						AND ((aBoxY[4] - aBoxY[2]- fPlasticVelo) >= cBoxWidth OR (aBoxY[4] - aBoxY[2]- fPlasticVelo) <= -cBoxWidth
								OR NOT (aBoxX[4] > cXforBox4OnPlasticBelt_min AND aBoxX[4] <= cXforBox4OnPlasticBelt_max));	
						
	aBoxPlasticBelt[3] := aBoxX[3] > cXforBox3OnPlasticBelt_min AND aBoxX[3] <= cXforBox3OnPlasticBelt_max										
						AND ((aBoxY[1] - aBoxY[3] - fPlasticVelo) >= cBoxWidth OR (aBoxY[1] - aBoxY[3] - fPlasticVelo) <= -cBoxWidth
								OR NOT (aBoxX[1] > cXforBox1OnPlasticBelt_min AND aBoxX[1] <= cXforBox1OnPlasticBelt_max))
						AND ((aBoxY[2] - aBoxY[3]- fPlasticVelo) >= cBoxWidth OR (aBoxY[2] - aBoxY[3]- fPlasticVelo) <= -cBoxWidth
								OR NOT (aBoxX[2] > cXforBox2OnPlasticBelt_min AND aBoxX[2] <= cXforBox2OnPlasticBelt_max))
						AND ((aBoxY[4] - aBoxY[3]- fPlasticVelo) >= cBoxWidth OR (aBoxY[4] - aBoxY[3]- fPlasticVelo) <= -cBoxWidth
								OR NOT (aBoxX[4] > cXforBox4OnPlasticBelt_min AND aBoxX[4] <= cXforBox4OnPlasticBelt_max));	
						
	aBoxPlasticBelt[4] := aBoxX[4] > cXforBox4OnPlasticBelt_min AND aBoxX[4] <= cXforBox4OnPlasticBelt_max										
						AND ((aBoxY[1] - aBoxY[4] - fPlasticVelo) >= cBoxWidth OR (aBoxY[1] - aBoxY[4] - fPlasticVelo) <= -cBoxWidth
								OR NOT (aBoxX[1] > cXforBox1OnPlasticBelt_min AND aBoxX[1] <= cXforBox1OnPlasticBelt_max))
						AND ((aBoxY[2] - aBoxY[4] - fPlasticVelo) >= cBoxWidth OR (aBoxY[2] - aBoxY[4] - fPlasticVelo) <= -cBoxWidth
								OR NOT (aBoxX[2] > cXforBox2OnPlasticBelt_min AND aBoxX[2] <= cXforBox2OnPlasticBelt_max))
						AND ((aBoxY[3] - aBoxY[4]- fPlasticVelo) >= cBoxWidth OR (aBoxY[3] - aBoxY[4]- fPlasticVelo) <= -cBoxWidth
								OR NOT (aBoxX[3] > cXforBox3OnPlasticBelt_min AND aBoxX[3] <= cXforBox3OnPlasticBelt_max));

// =========================================================
// Motion of boxes on metal belt and back to the start position number 4

	FOR nState := 1 TO 4 BY 1 DO	
		IF bPlasticAxisMoves THEN
				IF 	aBoxPlasticBelt[nState] THEN	
					// Check the state and direction of motion		
					IF bAuto OR bSemi OR (NOT bAuto AND bButtonPlasticFwIn) THEN
						// Move box to the end of metal belt and then back to position 4	
						IF aBoxY[nState] <= (cYBoxesOnMetalPlasticBelt_min + 0.1) AND aBoxY[nState] > cYBoxesOnMetalPlasticBelt_max THEN
							aBoxY[nState] := aBoxY[nState] + fPlasticVelo;
						END_IF
						
					ELSIF NOT bAuto AND bButtonPlasticBwIn THEN
						IF aBoxY[nState] + fPlasticVelo <= (cYBoxesOnMetalPlasticBelt_min - 0.1) THEN
							aBoxY[nState] := aBoxY[nState] + fPlasticVelo;
						END_IF
					END_IF
				END_IF
		END_IF
		
		IF aBoxY[nState] <= cYBoxesOnMetalPlasticBelt_max AND nLastBox = 0 THEN
			aBoxY[nState] := cYforAllBoxesStartPosMainBelt;
			aBoxX[nState] := cXforAllBoxesStartPosMainBelt + nState*cBoxWidth;
		END_IF
	END_FOR

// =========================================================
END_METHOD

METHOD PRIVATE AxisRotation
VAR_INPUT
END_VAR
// =========================================================
// Rotation of main axis
	
	fbTimerMainAxis(IN := bMainAxisMoves,
					PT := tMoveAxis);
	
	IF fbTimerMainAxis.Q THEN
		fbTimerMainAxis(IN := FALSE);
		
		IF bAuto OR bSemi THEN
			nAngleMain := nAngleMain + cAxisMovementSemiPlusAuto;
			
		ELSIF bButtonMainFwIn THEN
			nAngleMain := nAngleMain + cAxisMovementManual;
			
		ELSIF bButtonMainBwIn THEN
			nAngleMain := nAngleMain - cAxisMovementManual;
		END_IF
	END_IF

// =========================================================
// Rotation of metal axis
	
	fbTimerMetalAxis( 	IN := bMetalAxisMoves,
						PT := tMoveAxis);
	
	IF fbTimerMetalAxis.Q THEN
		fbTimerMetalAxis( IN := FALSE );
		
		IF bAuto OR bSemi THEN
			nAngleMetal := nAngleMetal + cAxisMovementSemiPlusAuto;
			
		ELSIF bButtonMetalFwIn THEN
			nAngleMetal := nAngleMetal + cAxisMovementManual;
			
		ELSIF bButtonMetalBwIn THEN
			nAngleMetal := nAngleMetal - cAxisMovementManual;
		END_IF
	END_IF

// =========================================================
// Rotation of plastic axis
	
	fbTimerPlasticAxis( IN := bPlasticAxisMoves,
						PT := tMoveAxis);
	
	IF fbTimerPlasticAxis.Q THEN
		fbTimerPlasticAxis( IN := FALSE );
		
		IF bAuto OR bSemi THEN
			nAnglePlastic := nAnglePlastic + cAxisMovementSemiPlusAuto;
			
		ELSIF bButtonPlasticFwIn THEN
			nAnglePlastic := nAnglePlastic + cAxisMovementManual;
			
		ELSIF bButtonPlasticBwIn THEN
			nAnglePlastic := nAnglePlastic - cAxisMovementManual;
		END_IF
	END_IF

// =========================================================
END_METHOD

METHOD PRIVATE Barrier_Clamp_Cyl
VAR_INPUT
END_VAR
// =========================================================
// Moving clamp cylinder
	
	IF bClampToWork THEN
		IF (fYClamp + cClampMovement) < cYClampCylEndPos THEN
			fYClamp := fYClamp + cClampMovement;
		ELSE
			fYClamp := cYClampCylEndPos;
		END_IF
		
	ELSE
		IF (fYClamp - cClampMovement) > cYClampCylStartPos THEN
			fYClamp := fYClamp - cClampMovement;
		ELSE
			fYClamp := cYClampCylStartPos;
		END_IF
	END_IF

// =========================================================
// =========================================================
// Moving barrier cylinder
	
	IF bBarrierToWork THEN
		IF (fYBarrier + cBarrierMovement) < cYBarrierCylEndPos THEN
			fYBarrier := fYBarrier + cBarrierMovement;
		ELSE
			fYBarrier := cYBarrierCylEndPos;
		END_IF
		
	ELSE
		IF (fYBarrier - cBarrierMovement) > cYBarrierCylStartPos THEN
			fYBarrier := fYBarrier - cBarrierMovement;
		ELSE
			fYBarrier := cYBarrierCylStartPos;
		END_IF
	END_IF

// =========================================================
// Checking position of boxes related to the barrier cylinder
	
	IF fYBarrier <= cBoxWidth AND NOT bBarrierToWork THEN
		FOR nState := 1 TO 4 BY 1 DO
			IF aBoxX[nState] > (-cBoxWidth + 0.11 + cBoxWidth*nState) AND aBoxX[nState] < (cBoxWidth*nState + cBarrierWidth) AND aBoxY[nState] = 0
			AND NOT bStopped THEN
				bAccident := TRUE;
			END_IF
		END_FOR
	END_IF

// =========================================================
END_METHOD

METHOD PRIVATE ButtonColors
VAR_INPUT
END_VAR
// =========================================================
// Start button
		
	IF (bAccident OR (bPowerEnabled AND (NOT bStarted OR (bSemi AND bStarted))
		AND NOT bButtonStopIn AND NOT bButtonAbortIn AND NOT bButtonResetIn
		AND (bAuto OR bSemi OR bManual OR bMaintenance))) AND NOT (bError AND bIdle) THEN
		
			IF bButtonStartOut THEN
				nButtonColorStart := cGreen;
			ELSE
				nButtonColorStart := cYellow;
			END_IF
			
			bButtonColorStart := TRUE;
	ELSE
		bButtonColorStart := FALSE;
	END_IF

// =========================================================
// Stop button
		
	IF (bStarted OR bIdle) AND (bAuto OR bSemi OR bManual OR bMaintenance) THEN
		IF bButtonStopOut THEN
			nButtonColorStop := cGreen;
		ELSE
			nButtonColorStop := cYellow;
		END_IF
		
		bButtonColorStop := TRUE;
	ELSE
		bButtonColorStop := FALSE;
	END_IF

// =========================================================
// Reset button
		
	IF bStopped AND bPowerEnabled THEN
		IF bButtonResetOut THEN
			nButtonColorReset := cGreen;
		ELSE
			nButtonColorReset := cYellow;		
		END_IF
		
		bButtonColorReset := TRUE;
	ELSE
		bButtonColorReset := FALSE;
	END_IF

// =========================================================
// Mode buttons
	
	IF bPowerEnabled THEN
		IF NOT bAuto THEN
			IF bIdle THEN
				nButtonColorAuto 	:= cYellow;
				bButtonColorAuto 	:= TRUE;
			ELSE
				bButtonColorAuto 	:= FALSE;
			END_IF
		ELSE
			nButtonColorAuto 		:= cGreen;
			bButtonColorAuto 		:= TRUE;
		END_IF
		
		IF NOT bSemi THEN
			IF bIdle THEN
				nButtonColorSemi 	:= cYellow;
				bButtonColorSemi 	:= TRUE;
			ELSE
				bButtonColorSemi 	:= FALSE;
			END_IF
		ELSE
			nButtonColorSemi 		:= cGreen;
			bButtonColorSemi 		:= TRUE;
		END_IF
		
		IF NOT bManual THEN
			IF bIdle THEN
				nButtonColorManu 	:= cYellow;
				bButtonColorManu 	:= TRUE;
			ELSE
				bButtonColorManu 	:= FALSE;
			END_IF
		ELSE
			nButtonColorManu 		:= cGreen;
			bButtonColorManu 		:= TRUE;
		END_IF
		
		IF NOT bMaintenance THEN
			IF bIdle THEN
				nButtonColorMaint 	:= cYellow;
				bButtonColorMaint 	:= TRUE;
			ELSE
				bButtonColorMaint 	:= FALSE;
			END_IF
		ELSE
			nButtonColorMaint 		:= cGreen;
			bButtonColorMaint 		:= TRUE;
		END_IF
	END_IF

// =========================================================
// Buttons to move cylinders and axes
			
	IF (bManual OR bMaintenance) AND bStarted THEN
	// Cylinders
		IF bButtonClampToWorkOut THEN
			nButtonColorClamp 	:= cPink;
		ELSE
			nButtonColorClamp 	:= cYellow;
		END_IF
		
		IF bButtonBarrierToWorkOut THEN
			nButtonColorBarrier := cPink;
		ELSE
			nButtonColorBarrier := cYellow;
		END_IF
		
		IF bButtonMetalToWorkOut THEN
			nButtonColorMetalCyl := cPink;
		ELSE
			nButtonColorMetalCyl := cYellow;
		END_IF
		
		IF bButtonPlasticToWorkOut THEN
			nButtonColorPlasticCyl := cPink;
		ELSE
			nButtonColorPlasticCyl := cYellow;
		END_IF
		
		bButtonColorClamp 		:= TRUE;
		bButtonColorBarrier 	:= TRUE;
		bButtonColorMetalCyl 	:= TRUE;
		bButtonColorPlasticCyl 	:= TRUE;
		
	// Axes
		IF bButtonMainBwOut THEN
			nButtonColorMainBw := cPink;
		ELSE
			nButtonColorMainBw := cYellow;
		END_IF
		
		IF bButtonMainFwOut THEN
			nButtonColorMainFw := cPink;
		ELSE
			nButtonColorMainFw := cYellow;
		END_IF
		
		IF bButtonMetalBwOut THEN
			nButtonColorMetalBw := cPink;
		ELSE
			nButtonColorMetalBw := cYellow;
		END_IF
		
		IF bButtonMetalFwOut THEN
			nButtonColorMetalFw := cPink;
		ELSE
			nButtonColorMetalFw := cYellow;
		END_IF
		
		IF bButtonPlasticBwOut THEN
			nButtonColorPlasticBw := cPink;
		ELSE
			nButtonColorPlasticBw := cYellow;
		END_IF
		
		IF bButtonPlasticFwOut THEN
			nButtonColorPlasticFw := cPink;
		ELSE
			nButtonColorPlasticFw := cYellow;
		END_IF
		
		bButtonColorMainBw 		:= NOT bButtonMainFwOut;
		bButtonColorMainFw 		:= NOT bButtonMainBwOut;
		bButtonColorMetalBw 	:= NOT bButtonMetalFwOut;
		bButtonColorMetalFw 	:= NOT bButtonMetalBwOut;
		bButtonColorPlasticBw 	:= NOT bButtonPlasticFwOut;
		bButtonColorPlasticFw 	:= NOT bButtonPlasticBwOut;
	ELSE
		bButtonColorClamp 		:= FALSE;
		bButtonColorBarrier 	:= FALSE;
		bButtonColorMetalCyl 	:= FALSE;
		bButtonColorPlasticCyl 	:= FALSE;
		bButtonColorMainBw 		:= FALSE;
		bButtonColorMainFw 		:= FALSE;
		bButtonColorMetalBw 	:= FALSE;
		bButtonColorMetalFw 	:= FALSE;
		bButtonColorPlasticBw 	:= FALSE;
		bButtonColorPlasticFw 	:= FALSE;
	END_IF
		
// =========================================================
// Button to control compressed air
			
	IF bMaintenance AND bStarted THEN
		IF bButtonComprAirIn THEN
			nButtonColorComprAir := cGreen;
		ELSE
			nButtonColorComprAir := cYellow;
		END_IF
		
		bButtonColorComprAir := TRUE;
	ELSE
		bButtonColorComprAir := FALSE;
	END_IF

// =========================================================
END_METHOD

METHOD PRIVATE ButtonSignals
VAR_INPUT
END_VAR
// =========================================================
// When machine is in requested state, buttons are turned off again

	IF bStartButtonOff THEN
		bButtonStartOut := FALSE;
	END_IF
	
	IF bStopped THEN
		bButtonStopOut := FALSE;
	END_IF
	
	IF bReset THEN
		bButtonResetOut := FALSE;
	END_IF
	
	IF bManual THEN
		bButtonManuOut := FALSE;
	END_IF
	
	IF bAuto THEN
		bButtonAutoOut := FALSE;
	END_IF
	
	IF bSemi THEN
		bButtonSemiOut := FALSE;
	END_IF
	
	IF bMaintenance THEN
		bButtonMaintenanceOut := FALSE;
	END_IF

// =========================================================
END_METHOD

METHOD PRIVATE CylinderMoveBoxes
VAR_INPUT
END_VAR
// =========================================================
// Metal cylinder - checking the positions of boxes
// bBoxMetalFree[1] is true, if any box blockades the movement of box 1 on metal belt
	
	aBoxMetalFree[1] := 	NOT (aBoxX[2] > cXforBox2OnMetalBelt_min AND aBoxX[2] <= cXforBox2OnMetalBelt_max AND (aBoxY[1] - aBoxY[2]) <= (cBoxWidth + 1))
						AND NOT (aBoxX[3] > cXforBox3OnMetalBelt_min AND aBoxX[3] <= cXforBox3OnMetalBelt_max AND (aBoxY[1] - aBoxY[3]) <= (cBoxWidth + 1))
						AND NOT (aBoxX[4] > cXforBox4OnMetalBelt_min AND aBoxX[4] <= cXforBox4OnMetalBelt_max AND (aBoxY[1] - aBoxY[4]) <= (cBoxWidth + 1));
	
	aBoxMetalFree[2] := 	NOT (aBoxX[1] > cXforBox1OnMetalBelt_min AND aBoxX[1] <= cXforBox1OnMetalBelt_max AND (aBoxY[2] - aBoxY[1]) <= (cBoxWidth + 1))
						AND NOT (aBoxX[3] > cXforBox3OnMetalBelt_min AND aBoxX[3] <= cXforBox3OnMetalBelt_max AND (aBoxY[2] - aBoxY[3]) <= (cBoxWidth + 1))
						AND NOT (aBoxX[4] > cXforBox4OnMetalBelt_min AND aBoxX[4] <= cXforBox4OnMetalBelt_max AND (aBoxY[2] - aBoxY[4]) <= (cBoxWidth + 1));
						
	aBoxMetalFree[3] := 	NOT (aBoxX[1] > cXforBox1OnMetalBelt_min AND aBoxX[1] <= cXforBox1OnMetalBelt_max AND (aBoxY[3] - aBoxY[1]) <= (cBoxWidth + 1))
						AND NOT (aBoxX[2] > cXforBox2OnMetalBelt_min AND aBoxX[2] <= cXforBox2OnMetalBelt_max AND (aBoxY[3] - aBoxY[2]) <= (cBoxWidth + 1))
						AND NOT (aBoxX[4] > cXforBox4OnMetalBelt_min AND aBoxX[4] <= cXforBox4OnMetalBelt_max AND (aBoxY[3] - aBoxY[4]) <= (cBoxWidth + 1));
						
	aBoxMetalFree[4] := 	NOT (aBoxX[1] > cXforBox1OnMetalBelt_min AND aBoxX[1] <= cXforBox1OnMetalBelt_max AND (aBoxY[4] - aBoxY[1]) <= (cBoxWidth + 1))
						AND NOT (aBoxX[2] > cXforBox2OnMetalBelt_min AND aBoxX[2] <= cXforBox2OnMetalBelt_max AND (aBoxY[4] - aBoxY[2]) <= (cBoxWidth + 1))
						AND NOT (aBoxX[3] > cXforBox3OnMetalBelt_min AND aBoxX[3] <= cXforBox3OnMetalBelt_max AND (aBoxY[4] - aBoxY[3]) <= (cBoxWidth + 1));

// =========================================================
// Metal cylinder - boxes motion
	
	FOR nState := 1 TO 4 BY 1 DO
		IF bMetalToWork AND aBoxMetalMove[nState] AND aBoxMetalFree[nState] THEN
			IF (fYMetal - cMetalPlasticCylMovement) >= (cYMetalPlasticCylEndPos + cMetalPlasticCylMovement) THEN
				fYMetal := fYMetal - cMetalPlasticCylMovement;
				
				IF (fYMetal - aBoxY[nState]) <= cYMetalPlasticCylOnMainBelt THEN
					aBoxY[nState] := aBoxY[nState] - cMetalPlasticCylMovement;
				END_IF
				
			ELSIF fYMetal = (cYMetalPlasticCylEndPos + cMetalPlasticCylMovement) AND (fYMetal - aBoxY[nState]) <= cYMetalPlasticCylOnMainBelt THEN
				aBoxY[nState] := aBoxY[nState] - 2*cMetalPlasticCylMovement;
				
			ELSE
				aBoxMetalMove[nState] := FALSE;
			END_IF
		END_IF	
	END_FOR

// =========================================================
// =========================================================
// Plastic cylinder - checking the positions of boxes

	aBoxPlasticFree[1] := 	NOT (aBoxX[2] > (cXforBox2OnPlasticBelt_min + 20) AND aBoxX[2] <= cXforBox2OnPlasticBelt_max AND (aBoxY[1] - aBoxY[2]) <= (cBoxWidth + 1))
						AND NOT (aBoxX[3] > (cXforBox3OnPlasticBelt_min + 20) AND aBoxX[3] <= cXforBox3OnPlasticBelt_max AND (aBoxY[1] - aBoxY[3]) <= (cBoxWidth + 1))
						AND NOT (aBoxX[4] > (cXforBox4OnPlasticBelt_min + 20) AND aBoxX[4] <= cXforBox4OnPlasticBelt_max AND (aBoxY[1] - aBoxY[4]) <= (cBoxWidth + 1));
	
	aBoxPlasticFree[2] := 	NOT (aBoxX[1] > (cXforBox1OnPlasticBelt_min + 20) AND aBoxX[1] <= cXforBox1OnPlasticBelt_max AND (aBoxY[2] - aBoxY[1]) <= (cBoxWidth + 1))
						AND NOT (aBoxX[3] > (cXforBox3OnPlasticBelt_min + 20) AND aBoxX[3] <= cXforBox3OnPlasticBelt_max AND (aBoxY[2] - aBoxY[3]) <= (cBoxWidth + 1))
						AND NOT (aBoxX[4] > (cXforBox4OnPlasticBelt_min + 20) AND aBoxX[4] <= cXforBox4OnPlasticBelt_max AND (aBoxY[2] - aBoxY[4]) <= (cBoxWidth + 1));
						
	aBoxPlasticFree[3] := 	NOT (aBoxX[1] > (cXforBox1OnPlasticBelt_min + 20) AND aBoxX[1] <= cXforBox1OnPlasticBelt_max AND (aBoxY[3] - aBoxY[1]) <= (cBoxWidth + 1))
						AND NOT (aBoxX[2] > (cXforBox2OnPlasticBelt_min + 20) AND aBoxX[2] <= cXforBox2OnPlasticBelt_max AND (aBoxY[3] - aBoxY[2]) <= (cBoxWidth + 1))
						AND NOT (aBoxX[4] > (cXforBox4OnPlasticBelt_min + 20) AND aBoxX[4] <= cXforBox4OnPlasticBelt_max AND (aBoxY[3] - aBoxY[4]) <= (cBoxWidth + 1));
						
	aBoxPlasticFree[4] := 	NOT (aBoxX[1] > (cXforBox1OnPlasticBelt_min + 20) AND aBoxX[1] <= cXforBox1OnPlasticBelt_max AND (aBoxY[4] - aBoxY[1]) <= (cBoxWidth + 1))
						AND NOT (aBoxX[2] > (cXforBox2OnPlasticBelt_min + 20) AND aBoxX[2] <= cXforBox2OnPlasticBelt_max AND (aBoxY[4] - aBoxY[2]) <= (cBoxWidth + 1))
						AND NOT (aBoxX[3] > (cXforBox3OnPlasticBelt_min + 20) AND aBoxX[3] <= cXforBox3OnPlasticBelt_max AND (aBoxY[4] - aBoxY[3]) <= (cBoxWidth + 1));
					
// =========================================================
// Plastic cylinder - boxes motion

	FOR nState := 1 TO 4 BY 1 DO
		IF bPlasticToWork AND aBoxPlasticMove[nState] AND aBoxPlasticFree[nState] THEN
			IF (fYPlastic - cMetalPlasticCylMovement) >= (cYMetalPlasticCylEndPos + cMetalPlasticCylMovement) THEN
				fYPlastic := fYPlastic - cMetalPlasticCylMovement;
				
				IF (fYPlastic - aBoxY[nState]) <= cYMetalPlasticCylOnMainBelt THEN
					aBoxY[nState] := aBoxY[nState] - cMetalPlasticCylMovement;
				END_IF
				
			ELSIF fYPlastic = (cYMetalPlasticCylEndPos + cMetalPlasticCylMovement) AND (fYPlastic - aBoxY[nState]) <= cYMetalPlasticCylOnMainBelt THEN
				aBoxY[nState] := aBoxY[nState] - 2*cMetalPlasticCylMovement;
				
			ELSE
				aBoxPlasticMove[nState] := FALSE;
			END_IF
		END_IF	
	END_FOR

// =========================================================
END_METHOD

METHOD PRIVATE ErrorMessages
VAR_INPUT
END_VAR
// =========================================================
// Error messages
	
	nMessages := 0;
		
	// Main axis
	IF nMainAxisErrorId = 0 THEN
		sMessageMainAxis 	:= '';
	ELSE
		nMessages 			:= nMessages + 1;
		sMessageMainAxis 	:= CONCAT('Error ID of main axis: ', UDINT_TO_STRING(nMainAxisErrorId));
	END_IF
	
	// Metal axis
	IF nMetalAxisErrorId = 0 THEN
		sMessageMetalAxis 	:= '';
	ELSE
		nMessages 			:= nMessages + 1;
		sMessageMetalAxis 	:= CONCAT('Error ID of metal axis: ', UDINT_TO_STRING(nMetalAxisErrorId));
	END_IF
	
	// Plastic axis
	IF nPlasticAxisErrorId = 0 THEN
		sMessagePlasticAxis	:= '';
	ELSE
		nMessages 			:= nMessages + 1;
		sMessagePlasticAxis	:= CONCAT('Error ID of plastic axis: ', UDINT_TO_STRING(nPlasticAxisErrorId));
	END_IF
	
	// Clamp cylinder
	IF bClampError THEN
		nMessages 			:= nMessages + 1;
		sMessageClamp 		:= CONCAT('Error of clamp cylinder: ', sClampErrMsg);
	ELSE
		sMessageClamp 		:= '';
	END_IF
	
	// Metal cylinder
	IF bMetalCylError THEN
		nMessages 			:= nMessages + 1;
		sMessageMetalCyl 	:= CONCAT('Error of metal cylinder: ', sMetalErrMsg);
	ELSE
		sMessageMetalCyl 	:= '';
	END_IF
	
	// Plastic cylinder
	IF bPlasticCylError THEN
		nMessages 			:= nMessages + 1;
		sMessagePlasticCyl 	:= CONCAT('Error of plastic cylinder: ', sPlasticErrMsg);
	ELSE
		sMessagePlasticCyl 	:= '';
	END_IF
	
// =========================================================
END_METHOD

METHOD PRIVATE LastBox
VAR_INPUT
END_VAR
// =========================================================
// Checking the last position on main belt
	
	IF 		(aBoxX[1] >= (cXforAllBoxesStartPosMainBelt + 1*cBoxWidth - 0.05))
	AND		(aBoxX[1] < (cXforAllBoxesStartPosMainBelt + 2*cBoxWidth - 0.05)) AND (aBoxY[1] = 0) THEN
		nLastBox := 1;
		
	ELSIF 	(aBoxX[2] >= (cXforAllBoxesStartPosMainBelt + 2*cBoxWidth - 0.05))
	AND 	(aBoxX[2] < (cXforAllBoxesStartPosMainBelt + 3*cBoxWidth - 0.05)) AND (aBoxY[2] = 0) THEN
		nLastBox := 2;	
		
	ELSIF 	(aBoxX[3] >= (cXforAllBoxesStartPosMainBelt + 3*cBoxWidth - 0.05))
	AND 	(aBoxX[3] < (cXforAllBoxesStartPosMainBelt + 4*cBoxWidth - 0.05)) AND (aBoxY[3] = 0) THEN
		nLastBox := 3;	
		
	ELSIF 	(aBoxX[4] >= cXforAllBoxesStartPosMainBelt + 4*cBoxWidth - 0.05)
	AND 	(aBoxX[4] < (cXforAllBoxesStartPosMainBelt + 5*cBoxWidth - 0.05)) AND (aBoxY[4] = 0) THEN
		nLastBox := 4;	
		
	ELSE
		nLastBox := 0;
	END_IF		

// =========================================================
END_METHOD

METHOD PRIVATE Metal_Plastic_Cyl
VAR_INPUT
END_VAR
// =========================================================
// Moving metal cylinder
	
	IF bMetalToWork THEN
		IF NOT (aBoxMetalMove[1] OR aBoxMetalMove[2] OR aBoxMetalMove[3] OR aBoxMetalMove[4]) THEN
			IF ((fYMetal - cMetalPlasticCylMovement) >= cYMetalPlasticCylEndPos) THEN
				fYMetal := fYMetal - cMetalPlasticCylMovement;
			END_IF
			
		ELSE
			FOR nState := 1 TO 4 BY 1 DO
				IF aBoxMetalMove[nState] THEN
					IF ((fYMetal - cMetalPlasticCylMovement) >= (aBoxY[nState] - cYMetalPlasticCylOnMainBelt - 0.1))
					AND ((fYMetal - cMetalPlasticCylMovement) >= cYMetalPlasticCylEndPos) THEN
						fYMetal := fYMetal - cMetalPlasticCylMovement;
					END_IF
				END_IF
			END_FOR
		END_IF
		
	ELSE
		IF ((fYMetal + cMetalPlasticCylMovement) < cYMetalPlasticCylStartPos) THEN
			fYMetal := fYMetal + cMetalPlasticCylMovement;
		ELSE
			fYMetal := cYMetalPlasticCylStartPos;
		END_IF
	END_IF

// =========================================================
// Checking position of boxes related to the metal cylinder
	
	IF (fYMetal < (cYMetalPlasticCylOnMainBelt + 0.1)) AND (fYMetal > (cYMetalPlasticCylOnMainBelt - 0.1)) AND bMetalToWork THEN
		FOR nState := 1 TO 4 BY 1 DO
			// box on main belt
			IF (aBoxY[nState] >= cYforAllBoxesOnMainBelt) THEN
				// box in right position related to the metal cylinder
				IF (aBoxX[nState] > (cXforAllBoxesCorrectPushMetalCyl_min + cBoxWidth*nState))
				AND (aBoxX[nState] <= (cXforAllBoxesCorrectPushMetalCyl_max + cBoxWidth*nState)) THEN
					aBoxMetalMove[nState] := TRUE;
				END_IF
				
				// box in wrong position related to the metal cylinder >> accident
				IF ((aBoxX[nState] > (cXforAllBoxesIncorrectPushMetalCyl_min + cBoxWidth*nState)
						AND aBoxX[nState] <= (cXforAllBoxesCorrectPushMetalCyl_min + cBoxWidth*nState))
					OR (aBoxX[nState] > (cXforAllBoxesCorrectPushMetalCyl_max + cBoxWidth*nState)
						AND aBoxX[nState] < (cXforAllBoxesIncorrectPushMetalCyl_max + cBoxWidth*nState)))
				AND NOT bStopped THEN
					bAccident := TRUE;
				END_IF
			END_IF
		END_FOR
	END_IF

// =========================================================
// =========================================================
// Moving plastic cylinder
	
	IF bPlasticToWork THEN
		IF NOT (aBoxPlasticMove[1] OR aBoxPlasticMove[2] OR aBoxPlasticMove[3] OR aBoxPlasticMove[4]) THEN
			IF ((fYPlastic - cMetalPlasticCylMovement) >= cYMetalPlasticCylEndPos) THEN
				fYPlastic := fYPlastic - cMetalPlasticCylMovement;
			END_IF
			
		ELSE
			FOR nState := 1 TO 4 BY 1 DO
				IF aBoxPlasticMove[nState] THEN
					IF ((fYPlastic - cMetalPlasticCylMovement) >= (aBoxY[nState] - cYMetalPlasticCylOnMainBelt - 0.1))
					AND ((fYPlastic - cMetalPlasticCylMovement) >= cYMetalPlasticCylEndPos) THEN
						fYPlastic := fYPlastic - cMetalPlasticCylMovement;
					END_IF
				END_IF
			END_FOR
		END_IF
		
	ELSE
		IF ((fYPlastic + cMetalPlasticCylMovement) < cYMetalPlasticCylStartPos) THEN
			fYPlastic := fYPlastic + cMetalPlasticCylMovement;
		ELSE
			fYPlastic := cYMetalPlasticCylStartPos;
		END_IF
	END_IF

// =========================================================
// Checking position of boxes related to the plastic cylinder
		
	IF ((aBoxX[1] > (cXforAllBoxesLastPossiblePosMainBelt + 1*cBoxWidth))
		OR (aBoxX[2] > (cXforAllBoxesLastPossiblePosMainBelt + 2*cBoxWidth))
		OR (aBoxX[3] > (cXforAllBoxesLastPossiblePosMainBelt + 3*cBoxWidth))
		OR (aBoxX[4] > (cXforAllBoxesLastPossiblePosMainBelt + 4*cBoxWidth)))
	AND NOT bStopped THEN
		bAccident := TRUE;
	END_IF
		
	IF (fYPlastic < (cYMetalPlasticCylOnMainBelt + 0.1)) AND (fYPlastic > (cYMetalPlasticCylOnMainBelt - 0.1)) AND bPlasticToWork THEN
		FOR nState := 1 TO 4 BY 1 DO
			// box on main belt
			IF aBoxY[nState] >= cYforAllBoxesOnMainBelt THEN
				// box in right position related to the plastic cylinder
				IF (aBoxX[nState] > (cXforAllBoxesCorrectPushPlasticCyl_min + cBoxWidth*nState))
				AND (aBoxX[nState] <= (cXforAllBoxesCorrectPushPlasticCyl_max + cBoxWidth*nState)) THEN
					aBoxPlasticMove[nState] := TRUE;
				END_IF
				
				// box in wrong position related to the plastic cylinder >> accident
				IF (aBoxX[nState] > (cXforAllBoxesIncorrectPushPlasticCyl_min + cBoxWidth*nState))
				AND (aBoxX[nState] <= (cXforAllBoxesCorrectPushPlasticCyl_min + cBoxWidth*nState))
				AND NOT bStopped THEN
					bAccident := TRUE;
				END_IF	
			END_IF
		END_FOR
	END_IF

// =========================================================
END_METHOD

METHOD PRIVATE Reset
VAR_INPUT
END_VAR
// =========================================================
// Resetting visu
	
	// Cylinder buttons
	bButtonClampToWorkOut 		:= FALSE;
	bButtonBarrierToWorkOut 	:= FALSE;
	bButtonMetalToWorkOut 		:= FALSE;
	bButtonPlasticToWorkOut 	:= FALSE;
	
	// Axis buttons
	bButtonMainBwOut 			:= FALSE;
	bButtonMainFwOut 			:= FALSE;
	bButtonMetalBwOut 			:= FALSE;
	bButtonMetalFwOut 			:= FALSE;
	bButtonPlasticBwOut			:= FALSE;
	bButtonPlasticFwOut			:= FALSE;
	
	// State and mode buttons
	bButtonStartOut 			:= FALSE;
	bButtonStopOut 				:= FALSE;
	bButtonResetOut 			:= FALSE;
	bButtonComprAirOut 			:= FALSE;
	bButtonManuOut 				:= FALSE;
	bButtonAutoOut 				:= FALSE;
	bButtonSemiOut 				:= FALSE;
	bButtonMaintenanceOut		:= FALSE;
	
	// Position of boxes and cylinders	
	FOR nState := 1 TO 4 BY 1 DO
		aBoxX[nState] 			:= 0;
		aBoxY[nState] 			:= 0;
		
		aBoxMetalMove[nState] 	:= FALSE;
		aBoxPlasticMove[nState]	:= FALSE;
		aBoxMainBelt[nState]	:= FALSE;
		aBoxMetalBelt[nState] 	:= FALSE;
		aBoxPlasticBelt[nState]	:= FALSE;
	END_FOR
	
	bAccident := FALSE;

// =========================================================
END_METHOD

END_FUNCTION_BLOCK

// ---- 00_Internal PackAL/POUs/PS_PackML_StateMachine_Auto.TcPOU
FUNCTION_BLOCK PS_PackML_StateMachine_Auto
VAR_INPUT
	Start				: BOOL;
	Hold				: BOOL;
	UnHold				: BOOL;
	Suspend				: BOOL;
	UnSuspend			: BOOL;
	Abort				: BOOL;
	Stop				: BOOL;
	Complete			: BOOL;
	Clear				: BOOL;
	Reset				: BOOL;
	StateComplete		: BOOL;
END_VAR
VAR_OUTPUT
	Status				: WORD;

	ST_Starting			: BOOL;
	ST_Completing		: BOOL;
	ST_Resetting		: BOOL;
	ST_Holding			: BOOL;
	ST_UnHolding		: BOOL;
	ST_Suspending		: BOOL;
	ST_UnSuspending		: BOOL;
	ST_Clearing			: BOOL;
	ST_Stopping			: BOOL;
	ST_Aborting			: BOOL;

	(* State Complete*)
	ST_Execute			: BOOL;
	ST_Complete			: BOOL;
	ST_Idle				: BOOL;
	ST_Held				: BOOL;
	ST_Suspended		: BOOL;
	ST_Stopped			: BOOL;
	ST_Aborted			: BOOL;

	(* additional *)
	Error				: BOOL;
	ErrorID				: DWORD;
	ePMLState			: E_PMLState := E_PMLState.IDLE;
END_VAR
VAR
	ePMLStatePrev		: E_PMLState;
	bStateChange		: BOOL;
	StateCompletePrev	: BOOL;
END_VAR

(* check for state change *)
IF ePMLStatePrev <> ePMLState THEN
	ePMLStatePrev 	:= ePMLState;
	bStateChange	:= TRUE;
ELSE
	bStateChange	:= FALSE;
END_IF


(* change to new state if requested *)
CASE ePMLState OF
	E_PMLState.UNDEFINED:
				(* undefined state *)
				IF bStateChange THEN
					(* transient state *)
					ST_Starting		:= FALSE;
					ST_Completing	:= FALSE;
					ST_Resetting	:= FALSE;
					ST_Holding		:= FALSE;
					ST_UnHolding	:= FALSE;
					ST_Suspending	:= FALSE;
					ST_UnSuspending	:= FALSE;
					ST_Clearing		:= FALSE;
					ST_Stopping		:= FALSE;
					ST_Aborting		:= FALSE;
		
					(* final state *)
					ST_Execute		:= FALSE;
					ST_Complete		:= FALSE;
					ST_Idle			:= FALSE;
					ST_Held			:= FALSE;
					ST_Suspended	:= FALSE;
					ST_Stopped		:= FALSE;
					ST_Aborted		:= FALSE;
				END_IF
		
				IF Abort THEN
					ePMLState 		:= E_PMLState.ABORTING;
					ST_Aborting		:= TRUE;
				ELSIF Stop THEN
					ePMLState 		:= E_PMLState.STOPPING;
					ST_Stopping		:= TRUE;
				END_IF


	E_PMLState.IDLE:
				(* final state *)
		
				IF bStateChange THEN
					(* transient state *)
					ST_Starting		:= FALSE;
					ST_Completing	:= FALSE;
					ST_Resetting	:= FALSE;
					ST_Holding		:= FALSE;
					ST_UnHolding	:= FALSE;
					ST_Suspending	:= FALSE;
					ST_UnSuspending	:= FALSE;
					ST_Clearing		:= FALSE;
					ST_Stopping		:= FALSE;
					ST_Aborting		:= FALSE;
		
					(* final state *)
					ST_Execute		:= FALSE;
					ST_Complete		:= FALSE;
					ST_Idle			:= TRUE;
					ST_Held			:= FALSE;
					ST_Suspended	:= FALSE;
					ST_Stopped		:= FALSE;
					ST_Aborted		:= FALSE;
				END_IF
		
				IF Abort THEN
					ePMLState 		:= E_PMLState.ABORTING;
					ST_Idle			:= FALSE;
					ST_Aborting		:= TRUE;
				ELSIF Stop THEN
					ePMLState 		:= E_PMLState.STOPPING;
					ST_Idle			:= FALSE;
					ST_Stopping		:= TRUE;
				ELSIF Start THEN
					ePMLState 		:= E_PMLState.STARTING;
					ST_Idle			:= FALSE;
					ST_Starting		:= TRUE;
				END_IF


	E_PMLState.STARTING:
				(* transient state *)
		
				IF bStateChange THEN
					(* transient state *)
					ST_Starting		:= TRUE;
					ST_Completing	:= FALSE;
					ST_Resetting	:= FALSE;
					ST_Holding		:= FALSE;
					ST_UnHolding	:= FALSE;
					ST_Suspending	:= FALSE;
					ST_UnSuspending	:= FALSE;
					ST_Clearing		:= FALSE;
					ST_Stopping		:= FALSE;
					ST_Aborting		:= FALSE;
		
					(* final state *)
					ST_Execute		:= FALSE;
					ST_Complete		:= FALSE;
					ST_Idle			:= FALSE;
					ST_Held			:= FALSE;
					ST_Suspended	:= FALSE;
					ST_Stopped		:= FALSE;
					ST_Aborted		:= FALSE;
				END_IF
		
				IF Abort THEN
					ePMLState 		:= E_PMLState.ABORTING;
					ST_Starting		:= FALSE;
					ST_Aborting		:= TRUE;
				ELSIF Stop THEN
					ePMLState 		:= E_PMLState.STOPPING;
					ST_Starting		:= FALSE;
					ST_Stopping		:= TRUE;
				ELSIF StateComplete AND NOT StateCompletePrev THEN
					ePMLState 		:= E_PMLState.EXECUTE;
					StateCompletePrev := StateComplete;
					ST_Starting		:= FALSE;
					ST_Execute		:= TRUE;
				END_IF


	E_PMLState.EXECUTE:
				(* final state *)
		
				IF bStateChange THEN
					(* transient state *)
					ST_Starting		:= FALSE;
					ST_Completing	:= FALSE;
					ST_Resetting	:= FALSE;
					ST_Holding		:= FALSE;
					ST_UnHolding	:= FALSE;
					ST_Suspending	:= FALSE;
					ST_UnSuspending	:= FALSE;
					ST_Clearing		:= FALSE;
					ST_Stopping		:= FALSE;
					ST_Aborting		:= FALSE;
		
					(* final state *)
					ST_Execute		:= TRUE;
					ST_Complete		:= FALSE;
					ST_Idle			:= FALSE;
					ST_Held			:= FALSE;
					ST_Suspended	:= FALSE;
					ST_Stopped		:= FALSE;
					ST_Aborted		:= FALSE;
				END_IF
		
				IF Abort THEN
					ePMLState 		:= E_PMLState.ABORTING;
					ST_Execute		:= FALSE;
					ST_Aborting		:= TRUE;
				ELSIF Stop THEN
					ePMLState 		:= E_PMLState.STOPPING;
					ST_Execute		:= FALSE;
					ST_Stopping		:= TRUE;
				ELSIF Suspend THEN
					ePMLState 		:= E_PMLState.SUSPENDING;
					ST_Execute		:= FALSE;
					ST_Suspending	:= TRUE;
				ELSIF Hold THEN
					ePMLState 		:= E_PMLState.HOLDING;
					ST_Execute		:= FALSE;
					ST_Holding		:= TRUE;
				ELSIF Complete THEN
					ePMLState 		:= E_PMLState.COMPLETING;
					ST_Execute		:= FALSE;
					ST_Completing	:= TRUE;
				END_IF


	E_PMLState.COMPLETING:
				(* transient state *)
		
				IF bStateChange THEN
					(* transient state *)
					ST_Starting		:= FALSE;
					ST_Completing	:= TRUE;
					ST_Resetting	:= FALSE;
					ST_Holding		:= FALSE;
					ST_UnHolding	:= FALSE;
					ST_Suspending	:= FALSE;
					ST_UnSuspending	:= FALSE;
					ST_Clearing		:= FALSE;
					ST_Stopping		:= FALSE;
					ST_Aborting		:= FALSE;
		
					(* final state *)
					ST_Execute		:= FALSE;
					ST_Complete		:= FALSE;
					ST_Idle			:= FALSE;
					ST_Held			:= FALSE;
					ST_Suspended	:= FALSE;
					ST_Stopped		:= FALSE;
					ST_Aborted		:= FALSE;
				END_IF
		
				IF Abort THEN
					ePMLState 		:= E_PMLState.ABORTING;
					ST_Completing	:= FALSE;
					ST_Aborting		:= TRUE;
				ELSIF Stop THEN
					ePMLState 		:= E_PMLState.STOPPING;
					ST_Completing	:= FALSE;
					ST_Stopping		:= TRUE;
				ELSIF StateComplete AND NOT StateCompletePrev THEN
					ePMLState 		:= E_PMLState.COMPLETE;
					StateCompletePrev := StateComplete;
					ST_Completing	:= FALSE;
					ST_Complete		:= TRUE;
				END_IF


	E_PMLState.COMPLETE:
				(* final state *)
		
				IF bStateChange THEN
					(* transient state *)
					ST_Starting		:= FALSE;
					ST_Completing	:= FALSE;
					ST_Resetting	:= FALSE;
					ST_Holding		:= FALSE;
					ST_UnHolding	:= FALSE;
					ST_Suspending	:= FALSE;
					ST_UnSuspending	:= FALSE;
					ST_Clearing		:= FALSE;
					ST_Stopping		:= FALSE;
					ST_Aborting		:= FALSE;
		
					(* final state *)
					ST_Execute		:= FALSE;
					ST_Complete		:= TRUE;
					ST_Idle			:= FALSE;
					ST_Held			:= FALSE;
					ST_Suspended	:= FALSE;
					ST_Stopped		:= FALSE;
					ST_Aborted		:= FALSE;
				END_IF
		
				IF Abort THEN
					ePMLState 		:= E_PMLState.ABORTING;
					ST_Complete		:= FALSE;
					ST_Aborting		:= TRUE;
				ELSIF Stop THEN
					ePMLState 		:= E_PMLState.STOPPING;
					ST_Complete		:= FALSE;
					ST_Stopping		:= TRUE;
				ELSIF Reset THEN
					ePMLState 		:= E_PMLState.RESETTING;
					ST_Complete		:= FALSE;
					ST_Resetting	:= TRUE;
				END_IF


	E_PMLState.RESETTING:
				(* transient state *)
		
				IF bStateChange THEN
					(* transient state *)
					ST_Starting		:= FALSE;
					ST_Completing	:= FALSE;
					ST_Resetting	:= TRUE;
					ST_Holding		:= FALSE;
					ST_UnHolding	:= FALSE;
					ST_Suspending	:= FALSE;
					ST_UnSuspending	:= FALSE;
					ST_Clearing		:= FALSE;
					ST_Stopping		:= FALSE;
					ST_Aborting		:= FALSE;
		
					(* final state *)
					ST_Execute		:= FALSE;
					ST_Complete		:= FALSE;
					ST_Idle			:= FALSE;
					ST_Held			:= FALSE;
					ST_Suspended	:= FALSE;
					ST_Stopped		:= FALSE;
					ST_Aborted		:= FALSE;
				END_IF
		
				IF Abort THEN
					ePMLState 		:= E_PMLState.ABORTING;
					ST_Resetting	:= FALSE;
					ST_Aborting		:= TRUE;
				ELSIF Stop THEN
					ePMLState 		:= E_PMLState.STOPPING;
					ST_Resetting	:= FALSE;
					ST_Stopping		:= TRUE;
				ELSIF StateComplete THEN
					ePMLState 		:= E_PMLState.IDLE;
					StateCompletePrev := StateComplete;
					ST_Resetting	:= FALSE;
					ST_Idle			:= TRUE;
				END_IF


	E_PMLState.HOLDING:
				(* transient state *)
		
				IF bStateChange THEN
					(* transient state *)
					ST_Starting		:= FALSE;
					ST_Completing	:= FALSE;
					ST_Resetting	:= FALSE;
					ST_Holding		:= TRUE;
					ST_UnHolding	:= FALSE;
					ST_Suspending	:= FALSE;
					ST_UnSuspending	:= FALSE;
					ST_Clearing		:= FALSE;
					ST_Stopping		:= FALSE;
					ST_Aborting		:= FALSE;
		
					(* final state *)
					ST_Execute		:= FALSE;
					ST_Complete		:= FALSE;
					ST_Idle			:= FALSE;
					ST_Held			:= FALSE;
					ST_Suspended	:= FALSE;
					ST_Stopped		:= FALSE;
					ST_Aborted		:= FALSE;
				END_IF
		
				IF Abort THEN
					ePMLState 		:= E_PMLState.ABORTING;
					ST_Holding		:= FALSE;
					ST_Aborting		:= TRUE;
				ELSIF Stop THEN
					ePMLState 		:= E_PMLState.STOPPING;
					ST_Holding		:= FALSE;
					ST_Stopping		:= TRUE;
				ELSIF StateComplete AND NOT StateCompletePrev THEN
					ePMLState 		:= E_PMLState.HELD;
					StateCompletePrev := StateComplete;
					ST_Holding		:= FALSE;
					ST_Held			:= TRUE;
				END_IF


	E_PMLState.HELD:
				(* final state *)

				IF bStateChange THEN
					(* transient state *)
					ST_Starting		:= FALSE;
					ST_Completing	:= FALSE;
					ST_Resetting	:= FALSE;
					ST_Holding		:= FALSE;
					ST_UnHolding	:= FALSE;
					ST_Suspending	:= FALSE;
					ST_UnSuspending	:= FALSE;
					ST_Clearing		:= FALSE;
					ST_Stopping		:= FALSE;
					ST_Aborting		:= FALSE;
		
					(* final state *)
					ST_Execute		:= FALSE;
					ST_Complete		:= FALSE;
					ST_Idle			:= FALSE;
					ST_Held			:= TRUE;
					ST_Suspended	:= FALSE;
					ST_Stopped		:= FALSE;
					ST_Aborted		:= FALSE;
				END_IF
		
				IF Abort THEN
					ePMLState 		:= E_PMLState.ABORTING;
					ST_Held			:= FALSE;
					ST_Aborting		:= TRUE;
				ELSIF Stop THEN
					ePMLState 		:= E_PMLState.STOPPING;
					ST_Held			:= FALSE;
					ST_Stopping		:= TRUE;
				ELSIF UnHold THEN
					ePMLState 		:= E_PMLState.UNHOLDING;
					ST_Held			:= FALSE;
					ST_UnHolding	:= TRUE;
				END_IF


	E_PMLState.UNHOLDING:
				(* transient state *)
		
				IF bStateChange THEN
					(* transient state *)
					ST_Starting		:= FALSE;
					ST_Completing	:= FALSE;
					ST_Resetting	:= FALSE;
					ST_Holding		:= FALSE;
					ST_UnHolding	:= TRUE;
					ST_Suspending	:= FALSE;
					ST_UnSuspending	:= FALSE;
					ST_Clearing		:= FALSE;
					ST_Stopping		:= FALSE;
					ST_Aborting		:= FALSE;
		
					(* final state *)
					ST_Execute		:= FALSE;
					ST_Complete		:= FALSE;
					ST_Idle			:= FALSE;
					ST_Held			:= FALSE;
					ST_Suspended	:= FALSE;
					ST_Stopped		:= FALSE;
					ST_Aborted		:= FALSE;
				END_IF
		
				IF Abort THEN
					ePMLState 		:= E_PMLState.ABORTING;
					ST_UnHolding	:= FALSE;
					ST_Aborting		:= TRUE;
				ELSIF Stop THEN
					ePMLState 		:= E_PMLState.STOPPING;
					ST_UnHolding	:= FALSE;
					ST_Stopping		:= TRUE;
				ELSIF StateComplete AND NOT StateCompletePrev THEN
					ePMLState 		:= E_PMLState.EXECUTE;
					StateCompletePrev := StateComplete;
					ST_UnHolding	:= FALSE;
					ST_Execute		:= TRUE;
				END_IF


	E_PMLState.SUSPENDING:
				(* transient state *)
		
				IF bStateChange THEN
					(* transient state *)
					ST_Starting		:= FALSE;
					ST_Completing	:= FALSE;
					ST_Resetting	:= FALSE;
					ST_Holding		:= FALSE;
					ST_UnHolding	:= FALSE;
					ST_Suspending	:= TRUE;
					ST_UnSuspending	:= FALSE;
					ST_Clearing		:= FALSE;
					ST_Stopping		:= FALSE;
					ST_Aborting		:= FALSE;
		
